KUKA KRL program: EPS_2_25694_GD01_A_20260114065858.src

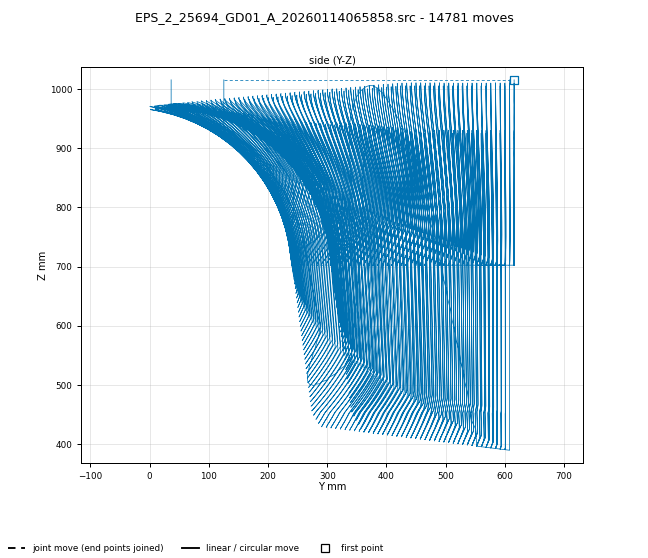
[picture p0: tool path of EPS_2_25694_GD01_A_20260114065858.src, 14781 of 14783 moves have a stored position in this frame; points joined in program order, loops and branches not executed]
&ACCESS RVP
&REL 4
&COMMENT QRS 19112012
&PARAM EDITMASK = *
DEF PART()
EXT BAS (BAS_COMMAND :IN,REAL :IN )
INT I
BAS (#INITMOV,0 )

;KUKA QRS Post kuka4.cps  Date:22-06-2017 !

File_ID=2969

QRS_PRE_INIT()

;Init var - Until changes are made in qrs_pre_init
Outlet_Square_prg=0
Inlet_1_Square_prg=0
Inlet_2_Square_prg=0
Inlet_3_Square_prg=0
Inlet_4_Square_prg=0
Inlet_5_Square_prg=0

Outlet_1={X 0.000, Y 425.000, Z 739.000, B 0.000, E1 0.000 }
Inlet_1={X 0.000, Y 466.000, Z 697.000, B 0.000, E1 153.000 }
Outlet_1_type=533
Inlet_1_type=457
;QRS#1=Sidecore dimensions
;QRS#2=525-21" Concrete
;QRS#3=450-18" Concrete
;QRS#4=
;QRS#5=
;QRS#6=
;QRS#7=
;QRS#8=
;QRS#9=S306-32
;QRS#10=28A PSX-2
;QRS#11=
;QRS#12=
;QRS#13=
;QRS#14=
;QRS#15=
;QRS#16=1220x127x1372 4,5'
;QRS#17=EPS Height
;QRS#18=1005,5
;QRS#19=*
;QRS#20= UPDATED VERSION 22-06-2017
;QRS#21=*
Outlet_Square=0250
Inlet_1_Square=0250
Inlet_2_Square=0
Inlet_3_Square=0
Inlet_4_Square=0
Inlet_5_Square=0
Mill_Square=1
Outlet_Square_Prg=263
Inlet_1_Square_prg=274

QRS_INIT()

$ADVANCE=5

; T1
PTP {E1 172.546,E2 172.546}
PTP {X 0,Y 615.562,A -85,B 0,C 180,E1 172.546,E2 172.546,E3 0,E4 0,E5 0,E6 0}
QRS_SPEED_INIT()
LIN {X 0,Y 615.562,Z 1015.5,A -85,B 0,C 180,E1 172.546,E2 172.546,E3 0,E4 0,E5 0,E6 0} C_VEL
LIN {X 0,Y 615.562,Z 704.53,A -85,B 0,C 180,E1 172.546,E2 172.546} C_VEL
LIN {X 0,Y 615.508,Z 702.53,A -85,B 0,C 180,E1 172.732,E2 172.732} C_VEL
LIN {X 0,Y 615.82,Z 702.53,A -85,B 0,C 180,E1 176.52,E2 176.52} C_VEL
LIN {X 0,Y 615.878,Z 702.53,A -85,B 0,C 180,E1 181.159,E2 181.159} C_VEL
LIN {X 0,Y 615.808,Z 702.53,A -85,B 0,C 180,E1 185.807,E2 185.807} C_VEL
LIN {X 0,Y 615.767,Z 702.53,A -85,B 0,C 180,E1 190.494,E2 190.494} C_VEL
LIN {X 0,Y 615.783,Z 702.53,A -85,B 0,C 180,E1 195.253,E2 195.253} C_VEL
LIN {X 0,Y 615.731,Z 702.53,A -85,B 0,C 180,E1 200.124,E2 200.124} C_VEL
LIN {X 0,Y 615.743,Z 702.53,A -85,B 0,C 180,E1 205.15,E2 205.15} C_VEL
LIN {X 0,Y 615.198,Z 702.53,A -85,B 0,C 180,E1 207.768,E2 207.768} C_VEL
LIN {X 0,Y 615.689,Z 702.53,A -85,B 0,C 180,E1 210.397,E2 210.397} C_VEL
LIN {X 0,Y 615.123,Z 702.53,A -85,B 0,C 180,E1 213.847,E2 213.847} C_VEL
LIN {X 0,Y 615.683,Z 702.53,A -85,B 0,C 180,E1 215.941,E2 215.941} C_VEL
LIN {X 0,Y 615.415,Z 702.53,A -85,B 0,C 180,E1 217.849,E2 217.849} C_VEL
LIN {X 0,Y 615.361,Z 702.53,A -85,B 0,C 180,E1 218.885,E2 218.885} C_VEL
LIN {X 0,Y 615.623,Z 702.53,A -85,B 0,C 180,E1 221.506,E2 221.506} C_VEL
LIN {X 0,Y 615.645,Z 702.53,A -85,B 0,C 180,E1 225.108,E2 225.108} C_VEL
LIN {X 0,Y 615.256,Z 702.53,A -85,B 0,C 180,E1 228.538,E2 228.538} C_VEL
LIN {X 0,Y 615.656,Z 702.53,A -85,B 0,C 180,E1 231.141,E2 231.141} C_VEL
LIN {X 0,Y 615.65,Z 702.53,A -85,B 0,C 180,E1 236.086,E2 236.086} C_VEL
LIN {X 0,Y 615.768,Z 702.53,A -85,B 0,C 180,E1 236.883,E2 236.883} C_VEL
LIN {X 0,Y 615.85,Z 702.53,A -85,B 0,C 180,E1 240.621,E2 240.621} C_VEL
LIN {X 0,Y 615.243,Z 702.53,A -85,B 0,C 180,E1 240.781,E2 240.781} C_VEL
LIN {X 0,Y 615.136,Z 702.999,A -85,B 0,C 180,E1 240.802,E2 240.802} C_VEL
LIN {X 0,Y 615.431,Z 753.05,A -85,B 0,C 180,E1 241.477,E2 241.477} C_VEL
LIN {X 0,Y 615.504,Z 764.124,A -85,B 0,C 180,E1 241.655,E2 241.655} C_VEL
LIN {X 0,Y 615.538,Z 778.609,A -85,B 0,C 180,E1 241.961,E2 241.961} C_VEL
LIN {X 0,Y 615.499,Z 788.804,A -85,B 0,C 180,E1 242.218,E2 242.218} C_VEL
LIN {X 0,Y 615.679,Z 804.599,A -85,B 0,C 180,E1 242.709,E2 242.709} C_VEL
LIN {X 0,Y 615.642,Z 817.021,A -85,B 0,C 180,E1 243.155,E2 243.155} C_VEL
LIN {X 0,Y 615.565,Z 826.938,A -85,B 0,C 180,E1 243.557,E2 243.557} C_VEL
LIN {X 0,Y 615.705,Z 842.65,A -85,B 0,C 180,E1 244.289,E2 244.289} C_VEL
LIN {X 0,Y 615.691,Z 854.983,A -85,B 0,C 180,E1 244.938,E2 244.938} C_VEL
LIN {X 0,Y 615.678,Z 866.612,A -85,B 0,C 180,E1 245.617,E2 245.617} C_VEL
LIN {X 0,Y 615.714,Z 878.424,A -85,B 0,C 180,E1 246.381,E2 246.381} C_VEL
LIN {X 0,Y 615.719,Z 889.118,A -85,B 0,C 180,E1 247.137,E2 247.137} C_VEL
LIN {X 0,Y 615.705,Z 900.424,A -85,B 0,C 180,E1 248.014,E2 248.014} C_VEL
LIN {X 0,Y 615.703,Z 909.682,A -85,B 0,C 180,E1 248.794,E2 248.794} C_VEL
LIN {X 0,Y 615.752,Z 919.817,A -85,B 0,C 180,E1 249.725,E2 249.725} C_VEL
LIN {X 0,Y 615.721,Z 929.079,A -85,B 0,C 180,E1 250.649,E2 250.649} C_VEL
LIN {X 0,Y 615.679,Z 937.435,A -85,B 0,C 180,E1 251.55,E2 251.55} C_VEL
LIN {X 0,Y 615.758,Z 945.796,A -85,B 0,C 180,E1 252.534,E2 252.534} C_VEL
LIN {X 0,Y 615.71,Z 953.699,A -85,B 0,C 180,E1 253.544,E2 253.544} C_VEL
LIN {X 0,Y 615.576,Z 960.443,A -85,B 0,C 180,E1 254.475,E2 254.475} C_VEL
LIN {X 0,Y 615.669,Z 968.075,A -85,B 0,C 180,E1 255.647,E2 255.647} C_VEL
LIN {X 0,Y 615.808,Z 973.451,A -85,B 0,C 180,E1 256.546,E2 256.546} C_VEL
LIN {X 0,Y 615.571,Z 979.922,A -85,B 0,C 180,E1 257.73,E2 257.73} C_VEL
LIN {X 0,Y 615.608,Z 985.635,A -85,B 0,C 180,E1 258.915,E2 258.915} C_VEL
LIN {X 0,Y 615.819,Z 990.644,A -85,B 0,C 180,E1 260.098,E2 260.098} C_VEL
LIN {X 0,Y 615.602,Z 995.072,A -85,B 0,C 180,E1 261.27,E2 261.27} C_VEL
LIN {X 0,Y 615.662,Z 999.448,A -85,B 0,C 180,E1 262.653,E2 262.653} C_VEL
LIN {X 0,Y 615.802,Z 1002.367,A -85,B 0,C 180,E1 263.749,E2 263.749} C_VEL
LIN {X 0,Y 615.545,Z 1005.385,A -85,B 0,C 180,E1 265.125,E2 265.125} C_VEL
LIN {X 0,Y 615.635,Z 1007.595,A -85,B 0,C 180,E1 266.521,E2 266.521} C_VEL
LIN {X 0,Y 615.819,Z 1008.672,A -85,B 0,C 180,E1 267.451,E2 267.451} C_VEL
LIN {X 0,Y 615.544,Z 1009.717,A -85,B 0,C 180,E1 268.842,E2 268.842} C_VEL
LIN {X 0,Y 615.843,Z 1009.658,A -85,B 0,C 180,E1 271.162,E2 271.162} C_VEL
LIN {X 0,Y 615.558,Z 1008.716,A -85,B 0,C 180,E1 272.555,E2 272.555} C_VEL
LIN {X 0,Y 615.598,Z 1006.932,A -85,B 0,C 180,E1 273.949,E2 273.949} C_VEL
LIN {X 0,Y 615.806,Z 1005.329,A -85,B 0,C 180,E1 274.878,E2 274.878} C_VEL
LIN {X 0,Y 615.606,Z 1002.401,A -85,B 0,C 180,E1 276.253,E2 276.253} C_VEL
LIN {X 0,Y 615.625,Z 999.259,A -85,B 0,C 180,E1 277.421,E2 277.421} C_VEL
LIN {X 0,Y 615.798,Z 995.025,A -85,B 0,C 180,E1 278.732,E2 278.732} C_VEL
LIN {X 0,Y 615.583,Z 990.661,A -85,B 0,C 180,E1 279.91,E2 279.91} C_VEL
LIN {X 0,Y 615.638,Z 985.611,A -85,B 0,C 180,E1 281.089,E2 281.089} C_VEL
LIN {X 0,Y 615.808,Z 979.871,A -85,B 0,C 180,E1 282.269,E2 282.269} C_VEL
LIN {X 0,Y 615.627,Z 973.442,A -85,B 0,C 180,E1 283.463,E2 283.463} C_VEL
LIN {X 0,Y 615.697,Z 966.18,A -85,B 0,C 180,E1 284.656,E2 284.656} C_VEL
LIN {X 0,Y 615.81,Z 960.631,A -85,B 0,C 180,E1 285.488,E2 285.488} C_VEL
LIN {X 0,Y 615.662,Z 951.188,A -85,B 0,C 180,E1 286.792,E2 286.792} C_VEL
LIN {X 0,Y 615.738,Z 942.596,A -85,B 0,C 180,E1 287.853,E2 287.853} C_VEL
LIN {X 0,Y 615.77,Z 934.395,A -85,B 0,C 180,E1 288.786,E2 288.786} C_VEL
LIN {X 0,Y 615.695,Z 924.501,A -85,B 0,C 180,E1 289.818,E2 289.818} C_VEL
LIN {X 0,Y 615.712,Z 916.513,A -85,B 0,C 180,E1 290.59,E2 290.59} C_VEL
LIN {X 0,Y 615.743,Z 906.008,A -85,B 0,C 180,E1 291.521,E2 291.521} C_VEL
LIN {X 0,Y 615.702,Z 896.053,A -85,B 0,C 180,E1 292.335,E2 292.335} C_VEL
LIN {X 0,Y 615.701,Z 886.27,A -85,B 0,C 180,E1 293.073,E2 293.073} C_VEL
LIN {X 0,Y 615.683,Z 874.62,A -85,B 0,C 180,E1 293.874,E2 293.874} C_VEL
LIN {X 0,Y 615.687,Z 862.583,A -85,B 0,C 180,E1 294.624,E2 294.624} C_VEL
LIN {X 0,Y 615.65,Z 851.845,A -85,B 0,C 180,E1 295.236,E2 295.236} C_VEL
LIN {X 0,Y 615.643,Z 840.977,A -85,B 0,C 180,E1 295.799,E2 295.799} C_VEL
LIN {X 0,Y 615.698,Z 826.817,A -85,B 0,C 180,E1 296.442,E2 296.442} C_VEL
LIN {X 0,Y 615.612,Z 813.606,A -85,B 0,C 180,E1 296.973,E2 296.973} C_VEL
LIN {X 0,Y 615.554,Z 804.458,A -85,B 0,C 180,E1 297.302,E2 297.302} C_VEL
LIN {X 0,Y 615.621,Z 787.798,A -85,B 0,C 180,E1 297.802,E2 297.802} C_VEL
LIN {X 0,Y 615.444,Z 775.356,A -85,B 0,C 180,E1 298.119,E2 298.119} C_VEL
LIN {X 0,Y 615.619,Z 763.086,A -85,B 0,C 180,E1 298.358,E2 298.358} C_VEL
LIN {X 0,Y 615.529,Z 741.859,A -85,B 0,C 180,E1 298.67,E2 298.67} C_VEL
LIN {X 0,Y 615.156,Z 705.781,A -85,B 0,C 180,E1 299.16,E2 299.16} C_VEL
LIN {X 0,Y 615.189,Z 702.53,A -85,B 0,C 180,E1 299.214,E2 299.214} C_VEL
LIN {X 0,Y 615.793,Z 702.53,A -85,B 0,C 180,E1 299.348,E2 299.348} C_VEL
LIN {X 0,Y 615.858,Z 702.53,A -85,B 0,C 180,E1 300.389,E2 300.389} C_VEL
LIN {X 0,Y 615.142,Z 702.53,A -85,B 0,C 180,E1 303.843,E2 303.843} C_VEL
LIN {X 0,Y 615.684,Z 702.53,A -85,B 0,C 180,E1 305.943,E2 305.943} C_VEL
LIN {X 0,Y 615.413,Z 702.53,A -85,B 0,C 180,E1 307.842,E2 307.842} C_VEL
LIN {X 0,Y 615.368,Z 702.53,A -85,B 0,C 180,E1 308.886,E2 308.886} C_VEL
LIN {X 0,Y 615.646,Z 702.53,A -85,B 0,C 180,E1 311.503,E2 311.503} C_VEL
LIN {X 0,Y 615.676,Z 702.53,A -85,B 0,C 180,E1 315.106,E2 315.106} C_VEL
LIN {X 0,Y 615.268,Z 702.53,A -85,B 0,C 180,E1 318.538,E2 318.538} C_VEL
LIN {X 0,Y 615.647,Z 702.53,A -85,B 0,C 180,E1 321.136,E2 321.136} C_VEL
LIN {X 0,Y 615.643,Z 702.53,A -85,B 0,C 180,E1 326.089,E2 326.089} C_VEL
LIN {X 0,Y 615.727,Z 702.53,A -85,B 0,C 180,E1 326.877,E2 326.877} C_VEL
LIN {X 0,Y 615.545,Z 702.53,A -85,B 0,C 180,E1 330.519,E2 330.519} C_VEL
LIN {X 0,Y 615.511,Z 702.53,A -85,B 0,C 180,E1 332.248,E2 332.248} C_VEL
LIN {X 0,Y 615.444,Z 702.53,A -85,B 0,C 180,E1 335.666,E2 335.666} C_VEL
LIN {X 0,Y 615.603,Z 702.53,A -85,B 0,C 180,E1 337.381,E2 337.381} C_VEL
LIN {X 0,Y 615.792,Z 702.53,A -85,B 0,C 180,E1 342.011,E2 342.011} C_VEL
LIN {X 0,Y 615.795,Z 702.53,A -85,B 0,C 180,E1 342.329,E2 342.329} C_VEL
LIN {X 0,Y 615.806,Z 702.53,A -85,B 0,C 180,E1 347.139,E2 347.139} C_VEL
LIN {X 0,Y 615.843,Z 702.53,A -85,B 0,C 180,E1 351.857,E2 351.857} C_VEL
LIN {X 0,Y 615.853,Z 702.53,A -85,B 0,C 180,E1 356.52,E2 356.52} C_VEL
LIN {X 0,Y 615.874,Z 702.53,A -85,B 0,C 180,E1 361.159,E2 361.159} C_VEL
LIN {X 0,Y 615.853,Z 702.53,A -85,B 0,C 180,E1 365.807,E2 365.807} C_VEL
LIN {X 0,Y 615.827,Z 702.53,A -85,B 0,C 180,E1 370.493,E2 370.493} C_VEL
LIN {X 0,Y 615.802,Z 702.53,A -85,B 0,C 180,E1 375.252,E2 375.252} C_VEL
LIN {X 0,Y 615.774,Z 702.53,A -85,B 0,C 180,E1 380.122,E2 380.122} C_VEL
LIN {X 0,Y 615.742,Z 702.53,A -85,B 0,C 180,E1 385.151,E2 385.151} C_VEL
LIN {X 0,Y 615.393,Z 702.53,A -85,B 0,C 180,E1 389.456,E2 389.456} C_VEL
LIN {X 0,Y 615.722,Z 702.53,A -85,B 0,C 180,E1 390.395,E2 390.395} C_VEL
LIN {X 0,Y 615.139,Z 702.53,A -85,B 0,C 180,E1 393.841,E2 393.841} C_VEL
LIN {X 0,Y 615.684,Z 702.53,A -85,B 0,C 180,E1 395.941,E2 395.941} C_VEL
LIN {X 0,Y 615.422,Z 702.53,A -85,B 0,C 180,E1 397.842,E2 397.842} C_VEL
LIN {X 0,Y 615.37,Z 702.53,A -85,B 0,C 180,E1 398.885,E2 398.885} C_VEL
LIN {X 0,Y 615.653,Z 702.53,A -85,B 0,C 180,E1 401.502,E2 401.502} C_VEL
LIN {X 0,Y 615.678,Z 702.53,A -85,B 0,C 180,E1 405.105,E2 405.105} C_VEL
LIN {X 0,Y 615.261,Z 702.53,A -85,B 0,C 180,E1 408.538,E2 408.538} C_VEL
LIN {X 0,Y 615.649,Z 702.53,A -85,B 0,C 180,E1 411.135,E2 411.135} C_VEL
LIN {X 0,Y 615.652,Z 702.53,A -85,B 0,C 180,E1 416.086,E2 416.086} C_VEL
LIN {X 0,Y 615.727,Z 702.53,A -85,B 0,C 180,E1 416.876,E2 416.876} C_VEL
LIN {X 0,Y 615.542,Z 702.53,A -85,B 0,C 180,E1 420.519,E2 420.519} C_VEL
LIN {X 0,Y 615.51,Z 702.53,A -85,B 0,C 180,E1 422.246,E2 422.246} C_VEL
LIN {X 0,Y 615.439,Z 702.53,A -85,B 0,C 180,E1 425.666,E2 425.666} C_VEL
LIN {X 0,Y 615.604,Z 702.53,A -85,B 0,C 180,E1 427.379,E2 427.379} C_VEL
LIN {X 0,Y 615.783,Z 702.53,A -85,B 0,C 180,E1 432.012,E2 432.012} C_VEL
LIN {X 0,Y 615.784,Z 702.53,A -85,B 0,C 180,E1 432.327,E2 432.327} C_VEL
LIN {X 0,Y 615.823,Z 702.53,A -85,B 0,C 180,E1 437.137,E2 437.137} C_VEL
LIN {X 0,Y 615.848,Z 702.53,A -85,B 0,C 180,E1 441.855,E2 441.855} C_VEL
LIN {X 0,Y 615.872,Z 702.53,A -85,B 0,C 180,E1 446.518,E2 446.518} C_VEL
LIN {X 0,Y 615.841,Z 702.53,A -85,B 0,C 180,E1 451.978,E2 451.978} C_VEL
LIN {X 0,Y 615.751,Z 702.53,A -85,B 0,C 180,E1 452.139,E2 452.139} C_VEL
LIN {X 0,Y 615.083,Z 702.53,A -85,B 0,C 180,E1 452.275,E2 452.275} C_VEL
LIN {X 0,Y 615.009,Z 702.774,A -85,B 0,C 180,E1 452.289,E2 452.289} C_VEL
LIN {X 0,Y 615.473,Z 717.375,A -85,B 0,C 180,E1 452.535,E2 452.535} C_VEL
LIN {X 0,Y 615.547,Z 729.182,A -85,B 0,C 180,E1 452.782,E2 452.782} C_VEL
LIN {X 0,Y 615.679,Z 740.947,A -85,B 0,C 180,E1 453.09,E2 453.09} C_VEL
LIN {X 0,Y 615.661,Z 751.951,A -85,B 0,C 180,E1 453.425,E2 453.425} C_VEL
LIN {X 0,Y 615.661,Z 761.787,A -85,B 0,C 180,E1 453.769,E2 453.769} C_VEL
LIN {X 0,Y 615.74,Z 774.534,A -85,B 0,C 180,E1 454.292,E2 454.292} C_VEL
LIN {X 0,Y 615.724,Z 784.661,A -85,B 0,C 180,E1 454.757,E2 454.757} C_VEL
LIN {X 0,Y 615.705,Z 794.885,A -85,B 0,C 180,E1 455.281,E2 455.281} C_VEL
LIN {X 0,Y 615.757,Z 806.034,A -85,B 0,C 180,E1 455.923,E2 455.923} C_VEL
LIN {X 0,Y 615.746,Z 815.383,A -85,B 0,C 180,E1 456.513,E2 456.513} C_VEL
LIN {X 0,Y 615.752,Z 824.921,A -85,B 0,C 180,E1 457.175,E2 457.175} C_VEL
LIN {X 0,Y 615.745,Z 833.623,A -85,B 0,C 180,E1 457.832,E2 457.832} C_VEL
LIN {X 0,Y 615.768,Z 842.678,A -85,B 0,C 180,E1 458.581,E2 458.581} C_VEL
LIN {X 0,Y 615.77,Z 850.852,A -85,B 0,C 180,E1 459.314,E2 459.314} C_VEL
LIN {X 0,Y 615.719,Z 859.842,A -85,B 0,C 180,E1 460.198,E2 460.198} C_VEL
LIN {X 0,Y 615.732,Z 866.741,A -85,B 0,C 180,E1 460.935,E2 460.935} C_VEL
LIN {X 0,Y 615.825,Z 874.318,A -85,B 0,C 180,E1 461.82,E2 461.82} C_VEL
LIN {X 0,Y 615.693,Z 881.358,A -85,B 0,C 180,E1 462.713,E2 462.713} C_VEL
LIN {X 0,Y 615.672,Z 887.77,A -85,B 0,C 180,E1 463.606,E2 463.606} C_VEL
LIN {X 0,Y 615.768,Z 892.697,A -85,B 0,C 180,E1 464.351,E2 464.351} C_VEL
LIN {X 0,Y 615.762,Z 898.133,A -85,B 0,C 180,E1 465.25,E2 465.25} C_VEL
LIN {X 0,Y 615.658,Z 904.637,A -85,B 0,C 180,E1 466.457,E2 466.457} C_VEL
LIN {X 0,Y 615.722,Z 908.539,A -85,B 0,C 180,E1 467.264,E2 467.264} C_VEL
LIN {X 0,Y 615.79,Z 911.864,A -85,B 0,C 180,E1 468.039,E2 468.039} C_VEL
LIN {X 0,Y 615.662,Z 915.248,A -85,B 0,C 180,E1 468.893,E2 468.893} C_VEL
LIN {X 0,Y 615.645,Z 917.494,A -85,B 0,C 180,E1 469.507,E2 469.507} C_VEL
LIN {X 0,Y 615.809,Z 921.259,A -85,B 0,C 180,E1 470.737,E2 470.737} C_VEL
LIN {X 0,Y 615.659,Z 924.082,A -85,B 0,C 180,E1 471.83,E2 471.83} C_VEL
LIN {X 0,Y 615.578,Z 925.81,A -85,B 0,C 180,E1 472.617,E2 472.617} C_VEL
LIN {X 0,Y 615.655,Z 927.35,A -85,B 0,C 180,E1 473.537,E2 473.537} C_VEL
LIN {X 0,Y 615.833,Z 928.448,A -85,B 0,C 180,E1 474.415,E2 474.415} C_VEL
LIN {X 0,Y 615.672,Z 929.19,A -85,B 0,C 180,E1 475.15,E2 475.15} C_VEL
LIN {X 0,Y 615.566,Z 929.862,A -85,B 0,C 180,E1 476.443,E2 476.443} C_VEL
LIN {X 0,Y 615.629,Z 929.941,A -85,B 0,C 180,E1 477.09,E2 477.09} C_VEL
LIN {X 0,Y 615.759,Z 929.762,A -85,B 0,C 180,E1 477.737,E2 477.737} C_VEL
LIN {X 0,Y 615.724,Z 929.269,A -85,B 0,C 180,E1 478.633,E2 478.633} C_VEL
LIN {X 0,Y 615.654,Z 928.477,A -85,B 0,C 180,E1 479.5,E2 479.5} C_VEL
LIN {X 0,Y 615.725,Z 927.304,A -85,B 0,C 180,E1 480.392,E2 480.392} C_VEL
LIN {X 0,Y 615.769,Z 925.725,A -85,B 0,C 180,E1 481.316,E2 481.316} C_VEL
LIN {X 0,Y 615.604,Z 923.699,A -85,B 0,C 180,E1 482.262,E2 482.262} C_VEL
LIN {X 0,Y 615.648,Z 920.259,A -85,B 0,C 180,E1 483.54,E2 483.54} C_VEL
LIN {X 0,Y 615.84,Z 917.349,A -85,B 0,C 180,E1 484.436,E2 484.436} C_VEL
LIN {X 0,Y 615.648,Z 912.677,A -85,B 0,C 180,E1 485.689,E2 485.689} C_VEL
LIN {X 0,Y 615.667,Z 908.205,A -85,B 0,C 180,E1 486.717,E2 486.717} C_VEL
LIN {X 0,Y 615.805,Z 904.101,A -85,B 0,C 180,E1 487.557,E2 487.557} C_VEL
LIN {X 0,Y 615.688,Z 898.359,A -85,B 0,C 180,E1 488.624,E2 488.624} C_VEL
LIN {X 0,Y 615.655,Z 891.34,A -85,B 0,C 180,E1 489.77,E2 489.77} C_VEL
LIN {X 0,Y 615.809,Z 884.46,A -85,B 0,C 180,E1 490.771,E2 490.771} C_VEL
LIN {X 0,Y 615.739,Z 877.668,A -85,B 0,C 180,E1 491.676,E2 491.676} C_VEL
LIN {X 0,Y 615.707,Z 871.255,A -85,B 0,C 180,E1 492.461,E2 492.461} C_VEL
LIN {X 0,Y 615.792,Z 862.791,A -85,B 0,C 180,E1 493.401,E2 493.401} C_VEL
LIN {X 0,Y 615.748,Z 855.188,A -85,B 0,C 180,E1 494.178,E2 494.178} C_VEL
LIN {X 0,Y 615.734,Z 846.42,A -85,B 0,C 180,E1 494.998,E2 494.998} C_VEL
LIN {X 0,Y 615.76,Z 839.129,A -85,B 0,C 180,E1 495.628,E2 495.628} C_VEL
LIN {X 0,Y 615.759,Z 830.678,A -85,B 0,C 180,E1 496.305,E2 496.305} C_VEL
LIN {X 0,Y 615.759,Z 821.705,A -85,B 0,C 180,E1 496.965,E2 496.965} C_VEL
LIN {X 0,Y 615.741,Z 811.832,A -85,B 0,C 180,E1 497.628,E2 497.628} C_VEL
LIN {X 0,Y 615.677,Z 800.964,A -85,B 0,C 180,E1 498.288,E2 498.288} C_VEL
LIN {X 0,Y 615.74,Z 791.443,A -85,B 0,C 180,E1 498.81,E2 498.81} C_VEL
LIN {X 0,Y 615.724,Z 780.829,A -85,B 0,C 180,E1 499.335,E2 499.335} C_VEL
LIN {X 0,Y 615.617,Z 771.032,A -85,B 0,C 180,E1 499.776,E2 499.776} C_VEL
LIN {X 0,Y 615.727,Z 759.41,A -85,B 0,C 180,E1 500.225,E2 500.225} C_VEL
LIN {X 0,Y 615.68,Z 746.955,A -85,B 0,C 180,E1 500.643,E2 500.643} C_VEL
LIN {X 0,Y 615.636,Z 737.302,A -85,B 0,C 180,E1 500.925,E2 500.925} C_VEL
LIN {X 0,Y 615.748,Z 724.036,A -85,B 0,C 180,E1 501.232,E2 501.232} C_VEL
LIN {X 0,Y 615.713,Z 712.712,A -85,B 0,C 180,E1 501.445,E2 501.445} C_VEL
LIN {X 0,Y 615.553,Z 702.53,A -85,B 0,C 180,E1 501.611,E2 501.611} C_VEL
LIN {X 0,Y 615.879,Z 702.53,A -85,B 0,C 180,E1 501.784,E2 501.784} C_VEL
LIN {X 0,Y 615.704,Z 702.53,A -85,B 0,C 180,E1 504.06,E2 504.06} C_VEL
LIN {X 0,Y 615.141,Z 702.53,A -85,B 0,C 180,E1 506.841,E2 506.841} C_VEL
LIN {X 0,Y 615.715,Z 702.53,A -85,B 0,C 180,E1 509.604,E2 509.604} C_VEL
LIN {X 0,Y 615.223,Z 702.53,A -85,B 0,C 180,E1 512.234,E2 512.234} C_VEL
LIN {X 0,Y 615.765,Z 702.53,A -85,B 0,C 180,E1 514.851,E2 514.851} C_VEL
LIN {X 0,Y 615.778,Z 702.53,A -85,B 0,C 180,E1 519.878,E2 519.878} C_VEL
LIN {X 0,Y 615.518,Z 702.53,A -85,B 0,C 180,E1 522.321,E2 522.321} C_VEL
LIN {X 0,Y 615.631,Z 702.53,A -85,B 0,C 180,E1 524.743,E2 524.743} C_VEL
LIN {X 0,Y 615.831,Z 702.53,A -85,B 0,C 180,E1 527.139,E2 527.139} C_VEL
LIN {X 0,Y 615.803,Z 702.53,A -85,B 0,C 180,E1 531.857,E2 531.857} C_VEL
LIN {X 0,Y 615.508,Z 702.53,A -85,B 0,C 180,E1 532.732,E2 532.732} C_VEL
LIN {X 0,Y 611.504,Z 702.53,A -85,B 0,C 180,E1 534.32,E2 534.32} C_VEL
LIN {X 0,Y 607.646,Z 702.53,A -85,B 0,C 180,E1 535.927,E2 535.927} C_VEL
LIN {X 0,Y 607.882,Z 702.53,A -85,B 0,C 180,E1 541.434,E2 541.434} C_VEL
LIN {X 0,Y 607.632,Z 702.53,A -85,B 0,C 180,E1 546.594,E2 546.594} C_VEL
LIN {X 0,Y 607.527,Z 702.53,A -85,B 0,C 180,E1 551.47,E2 551.47} C_VEL
LIN {X 0,Y 607.63,Z 702.53,A -85,B 0,C 180,E1 555.862,E2 555.862} C_VEL
LIN {X 0,Y 607.744,Z 702.53,A -85,B 0,C 180,E1 560.349,E2 560.349} C_VEL
LIN {X 0,Y 607.769,Z 702.53,A -85,B 0,C 180,E1 564.973,E2 564.973} C_VEL
LIN {X 0,Y 607.567,Z 702.53,A -85,B 0,C 180,E1 569.79,E2 569.79} C_VEL
LIN {X 0,Y 607.62,Z 702.53,A -85,B 0,C 180,E1 576.591,E2 576.591} C_VEL
LIN {X 0,Y 607.565,Z 702.53,A -85,B 0,C 180,E1 582.117,E2 582.117} C_VEL
LIN {X 0,Y 607.258,Z 702.53,A -85,B 0,C 180,E1 587.86,E2 587.86} C_VEL
LIN {X 0,Y 607.289,Z 702.53,A -85,B 0,C 180,E1 592.671,E2 592.671} C_VEL
LIN {X 0,Y 607.695,Z 702.53,A -85,B 0,C 180,E1 597.595,E2 597.595} C_VEL
LIN {X 0,Y 607.882,Z 702.53,A -85,B 0,C 180,E1 600.411,E2 600.411} C_VEL
LIN {X 0,Y 608.572,Z 775.577,A -85,B 0,C 180,E1 601.539,E2 601.539} C_VEL
LIN {X 0,Y 608.562,Z 814.928,A -85,B 0,C 180,E1 602.736,E2 602.736} C_VEL
LIN {X 0,Y 608.415,Z 852.42,A -85,B 0,C 180,E1 604.472,E2 604.472} C_VEL
LIN {X 0,Y 608.266,Z 888.674,A -85,B 0,C 180,E1 606.806,E2 606.806} C_VEL
LIN {X 0,Y 608.119,Z 920.038,A -85,B 0,C 180,E1 609.481,E2 609.481} C_VEL
LIN {X 0,Y 608.016,Z 947.232,A -85,B 0,C 180,E1 612.486,E2 612.486} C_VEL
LIN {X 0,Y 607.884,Z 970.252,A -85,B 0,C 180,E1 615.81,E2 615.81} C_VEL
LIN {X 0,Y 607.811,Z 987.976,A -85,B 0,C 180,E1 619.268,E2 619.268} C_VEL
LIN {X 0,Y 607.799,Z 1000.677,A -85,B 0,C 180,E1 622.869,E2 622.869} C_VEL
LIN {X 0,Y 607.67,Z 1006.955,A -85,B 0,C 180,E1 625.727,E2 625.727} C_VEL
LIN {X 0,Y 607.699,Z 1010.085,A -85,B 0,C 180,E1 628.577,E2 628.577} C_VEL
LIN {X 0,Y 607.885,Z 1010.086,A -85,B 0,C 180,E1 631.422,E2 631.422} C_VEL
LIN {X 0,Y 607.905,Z 1005.757,A -85,B 0,C 180,E1 634.984,E2 634.984} C_VEL
LIN {X 0,Y 607.892,Z 995.072,A -85,B 0,C 180,E1 638.925,E2 638.925} C_VEL
LIN {X 0,Y 607.908,Z 979.45,A -85,B 0,C 180,E1 642.545,E2 642.545} C_VEL
LIN {X 0,Y 607.957,Z 958.349,A -85,B 0,C 180,E1 646.03,E2 646.03} C_VEL
LIN {X 0,Y 608.033,Z 932.214,A -85,B 0,C 180,E1 649.268,E2 649.268} C_VEL
LIN {X 0,Y 608.17,Z 902.022,A -85,B 0,C 180,E1 652.138,E2 652.138} C_VEL
LIN {X 0,Y 608.309,Z 868.887,A -85,B 0,C 180,E1 654.552,E2 654.552} C_VEL
LIN {X 0,Y 608.48,Z 832.739,A -85,B 0,C 180,E1 656.513,E2 656.513} C_VEL
LIN {X 0,Y 608.589,Z 795.74,A -85,B 0,C 180,E1 657.917,E2 657.917} C_VEL
LIN {X 0,Y 608.661,Z 760.101,A -85,B 0,C 180,E1 658.759,E2 658.759} C_VEL
LIN {X 0,Y 607.904,Z 702.53,A -85,B 0,C 180,E1 659.587,E2 659.587} C_VEL
LIN {X 0,Y 607.619,Z 702.53,A -85,B 0,C 180,E1 666.587,E2 666.587} C_VEL
LIN {X 0,Y 607.606,Z 702.53,A -85,B 0,C 180,E1 672.11,E2 672.11} C_VEL
LIN {X 0,Y 607.275,Z 702.53,A -85,B 0,C 180,E1 677.858,E2 677.858} C_VEL
LIN {X 0,Y 607.28,Z 702.53,A -85,B 0,C 180,E1 682.671,E2 682.671} C_VEL
LIN {X 0,Y 607.588,Z 702.53,A -85,B 0,C 180,E1 687.611,E2 687.611} C_VEL
LIN {X 0,Y 607.59,Z 702.53,A -85,B 0,C 180,E1 691.837,E2 691.837} C_VEL
LIN {X 0,Y 607.473,Z 702.53,A -85,B 0,C 180,E1 698.116,E2 698.116} C_VEL
LIN {X 0,Y 607.777,Z 702.53,A -85,B 0,C 180,E1 702.658,E2 702.658} C_VEL
LIN {X 0,Y 607.875,Z 702.53,A -85,B 0,C 180,E1 707.081,E2 707.081} C_VEL
LIN {X 0,Y 607.617,Z 702.53,A -85,B 0,C 180,E1 712.857,E2 712.857} C_VEL
LIN {X 0,Y 607.732,Z 702.53,A -85,B 0,C 180,E1 717.143,E2 717.143} C_VEL
LIN {X 0,Y 607.869,Z 702.53,A -85,B 0,C 180,E1 721.411,E2 721.411} C_VEL
LIN {X 0,Y 607.675,Z 702.53,A -85,B 0,C 180,E1 726.632,E2 726.632} C_VEL
LIN {X 0,Y 607.598,Z 702.53,A -85,B 0,C 180,E1 731.446,E2 731.446} C_VEL
LIN {X 0,Y 607.677,Z 702.53,A -85,B 0,C 180,E1 735.837,E2 735.837} C_VEL
LIN {X 0,Y 607.78,Z 702.53,A -85,B 0,C 180,E1 740.323,E2 740.323} C_VEL
LIN {X 0,Y 607.769,Z 702.53,A -85,B 0,C 180,E1 744.948,E2 744.948} C_VEL
LIN {X 0,Y 607.595,Z 702.53,A -85,B 0,C 180,E1 749.762,E2 749.762} C_VEL
LIN {X 0,Y 607.624,Z 702.53,A -85,B 0,C 180,E1 756.562,E2 756.562} C_VEL
LIN {X 0,Y 607.609,Z 702.53,A -85,B 0,C 180,E1 762.082,E2 762.082} C_VEL
LIN {X 0,Y 607.29,Z 702.53,A -85,B 0,C 180,E1 767.863,E2 767.863} C_VEL
LIN {X 0,Y 607.288,Z 702.53,A -85,B 0,C 180,E1 772.633,E2 772.633} C_VEL
LIN {X 0,Y 607.599,Z 702.53,A -85,B 0,C 180,E1 777.567,E2 777.567} C_VEL
LIN {X 0,Y 607.58,Z 702.53,A -85,B 0,C 180,E1 781.843,E2 781.843} C_VEL
LIN {X 0,Y 607.491,Z 702.53,A -85,B 0,C 180,E1 788.124,E2 788.124} C_VEL
LIN {X 0,Y 607.741,Z 702.53,A -85,B 0,C 180,E1 792.665,E2 792.665} C_VEL
LIN {X 0,Y 607.896,Z 702.53,A -85,B 0,C 180,E1 797.091,E2 797.091} C_VEL
LIN {X 0,Y 607.622,Z 702.53,A -85,B 0,C 180,E1 802.867,E2 802.867} C_VEL
LIN {X 0,Y 607.686,Z 702.53,A -85,B 0,C 180,E1 807.153,E2 807.153} C_VEL
LIN {X 0,Y 607.944,Z 702.53,A -85,B 0,C 180,E1 811.956,E2 811.956} C_VEL
LIN {X 0,Y 608.422,Z 742.827,A -85,B 0,C 180,E1 812.843,E2 812.843} C_VEL
LIN {X 0,Y 608.35,Z 776.479,A -85,B 0,C 180,E1 814.09,E2 814.09} C_VEL
LIN {X 0,Y 608.247,Z 809.586,A -85,B 0,C 180,E1 815.874,E2 815.874} C_VEL
LIN {X 0,Y 608.108,Z 841.848,A -85,B 0,C 180,E1 818.266,E2 818.266} C_VEL
LIN {X 0,Y 607.975,Z 869.921,A -85,B 0,C 180,E1 821.091,E2 821.091} C_VEL
LIN {X 0,Y 607.93,Z 892.853,A -85,B 0,C 180,E1 824.189,E2 824.189} C_VEL
LIN {X 0,Y 607.864,Z 909.669,A -85,B 0,C 180,E1 827.332,E2 827.332} C_VEL
LIN {X 0,Y 607.936,Z 921.864,A -85,B 0,C 180,E1 830.715,E2 830.715} C_VEL
LIN {X 0,Y 607.78,Z 927.704,A -85,B 0,C 180,E1 833.407,E2 833.407} C_VEL
LIN {X 0,Y 607.708,Z 930.443,A -85,B 0,C 180,E1 836.681,E2 836.681} C_VEL
LIN {X 0,Y 607.783,Z 928.711,A -85,B 0,C 180,E1 839.773,E2 839.773} C_VEL
LIN {X 0,Y 607.739,Z 922.093,A -85,B 0,C 180,E1 843.111,E2 843.111} C_VEL
LIN {X 0,Y 607.795,Z 911.669,A -85,B 0,C 180,E1 846.109,E2 846.109} C_VEL
LIN {X 0,Y 607.806,Z 895.517,A -85,B 0,C 180,E1 849.279,E2 849.279} C_VEL
LIN {X 0,Y 607.951,Z 874.115,A -85,B 0,C 180,E1 852.321,E2 852.321} C_VEL
LIN {X 0,Y 608.077,Z 847.473,A -85,B 0,C 180,E1 855.139,E2 855.139} C_VEL
LIN {X 0,Y 608.19,Z 817.921,A -85,B 0,C 180,E1 857.487,E2 857.487} C_VEL
LIN {X 0,Y 608.323,Z 784.262,A -85,B 0,C 180,E1 859.458,E2 859.458} C_VEL
LIN {X 0,Y 608.402,Z 747.231,A -85,B 0,C 180,E1 860.936,E2 860.936} C_VEL
LIN {X 0,Y 608.502,Z 711.075,A -85,B 0,C 180,E1 861.78,E2 861.78} C_VEL
LIN {X 0,Y 607.958,Z 702.53,A -85,B 0,C 180,E1 861.946,E2 861.946} C_VEL
LIN {X 0,Y 607.444,Z 702.53,A -85,B 0,C 180,E1 868.576,E2 868.576} C_VEL
LIN {X 0,Y 607.422,Z 702.53,A -85,B 0,C 180,E1 873.457,E2 873.457} C_VEL
LIN {X 0,Y 607.315,Z 702.53,A -85,B 0,C 180,E1 876.833,E2 876.833} C_VEL
LIN {X 0,Y 607.631,Z 702.53,A -85,B 0,C 180,E1 881.181,E2 881.181} C_VEL
LIN {X 0,Y 607.936,Z 702.53,A -85,B 0,C 180,E1 887.106,E2 887.106} C_VEL
LIN {X 0,Y 607.586,Z 702.53,A -85,B 0,C 180,E1 892.88,E2 892.88} C_VEL
LIN {X 0,Y 607.646,Z 702.53,A -85,B 0,C 180,E1 895.927,E2 895.927} C_VEL
LIN {X 0,Y 606.323,Z 702.53,A -85,B 0,C 180,E1 896.741,E2 896.741} C_VEL
LIN {X 0,Y 599.65,Z 702.53,A -85,B 0,C 180,E1 898.952,E2 898.952} C_VEL
LIN {X 0,Y 599.573,Z 702.53,A -85,B 0,C 180,E1 899.162,E2 899.162} C_VEL
LIN {X 0,Y 599.624,Z 702.53,A -85,B 0,C 180,E1 902.896,E2 902.896} C_VEL
LIN {X 0,Y 599.58,Z 702.53,A -85,B 0,C 180,E1 907.239,E2 907.239} C_VEL
LIN {X 0,Y 599.601,Z 702.53,A -85,B 0,C 180,E1 911.624,E2 911.624} C_VEL
LIN {X 0,Y 599.473,Z 702.53,A -85,B 0,C 180,E1 916.95,E2 916.95} C_VEL
LIN {X 0,Y 599.53,Z 702.53,A -85,B 0,C 180,E1 921.362,E2 921.362} C_VEL
LIN {X 0,Y 599.742,Z 702.53,A -85,B 0,C 180,E1 925.331,E2 925.331} C_VEL
LIN {X 0,Y 599.488,Z 702.53,A -85,B 0,C 180,E1 931.146,E2 931.146} C_VEL
LIN {X 0,Y 599.652,Z 702.53,A -85,B 0,C 180,E1 937.158,E2 937.158} C_VEL
LIN {X 0,Y 599.551,Z 702.53,A -85,B 0,C 180,E1 943.121,E2 943.121} C_VEL
LIN {X 0,Y 599.409,Z 702.53,A -85,B 0,C 180,E1 949.114,E2 949.114} C_VEL
LIN {X 0,Y 599.307,Z 702.53,A -85,B 0,C 180,E1 953.683,E2 953.683} C_VEL
LIN {X 0,Y 599.74,Z 702.53,A -85,B 0,C 180,E1 958.103,E2 958.103} C_VEL
LIN {X 0,Y 599.864,Z 702.564,A -85,B 0,C 180,E1 959.978,E2 959.978} C_VEL
LIN {X 0,Y 601.417,Z 710.419,A -85,B 0,C 180,E1 960.169,E2 960.169} C_VEL
LIN {X 0,Y 601.6,Z 776.602,A -85,B 0,C 180,E1 961.201,E2 961.201} C_VEL
LIN {X 0,Y 601.474,Z 815.69,A -85,B 0,C 180,E1 962.416,E2 962.416} C_VEL
LIN {X 0,Y 601.133,Z 854.192,A -85,B 0,C 180,E1 964.241,E2 964.241} C_VEL
LIN {X 0,Y 600.768,Z 889.761,A -85,B 0,C 180,E1 966.585,E2 966.585} C_VEL
LIN {X 0,Y 600.495,Z 920.701,A -85,B 0,C 180,E1 969.276,E2 969.276} C_VEL
LIN {X 0,Y 600.272,Z 948.698,A -85,B 0,C 180,E1 972.442,E2 972.442} C_VEL
LIN {X 0,Y 600.065,Z 971.361,A -85,B 0,C 180,E1 975.809,E2 975.809} C_VEL
LIN {X 0,Y 599.955,Z 988.886,A -85,B 0,C 180,E1 979.343,E2 979.343} C_VEL
LIN {X 0,Y 599.899,Z 1000.677,A -85,B 0,C 180,E1 982.774,E2 982.774} C_VEL
LIN {X 0,Y 599.767,Z 1006.955,A -85,B 0,C 180,E1 985.671,E2 985.671} C_VEL
LIN {X 0,Y 599.8,Z 1010.086,A -85,B 0,C 180,E1 988.558,E2 988.558} C_VEL
LIN {X 0,Y 599.978,Z 1010.086,A -85,B 0,C 180,E1 991.441,E2 991.441} C_VEL
LIN {X 0,Y 599.993,Z 1005.757,A -85,B 0,C 180,E1 995.05,E2 995.05} C_VEL
LIN {X 0,Y 599.99,Z 995.073,A -85,B 0,C 180,E1 999.044,E2 999.044} C_VEL
LIN {X 0,Y 600.043,Z 979.451,A -85,B 0,C 180,E1 1002.712,E2 1002.712} C_VEL
LIN {X 0,Y 600.116,Z 957.721,A -85,B 0,C 180,E1 1006.333,E2 1006.333} C_VEL
LIN {X 0,Y 600.355,Z 932.069,A -85,B 0,C 180,E1 1009.541,E2 1009.541} C_VEL
LIN {X 0,Y 600.638,Z 901.462,A -85,B 0,C 180,E1 1012.478,E2 1012.478} C_VEL
LIN {X 0,Y 600.985,Z 866.931,A -85,B 0,C 180,E1 1014.999,E2 1014.999} C_VEL
LIN {X 0,Y 601.369,Z 828.903,A -85,B 0,C 180,E1 1017.033,E2 1017.033} C_VEL
LIN {X 0,Y 601.58,Z 789.536,A -85,B 0,C 180,E1 1018.464,E2 1018.464} C_VEL
LIN {X 0,Y 601.785,Z 750.404,A -85,B 0,C 180,E1 1019.273,E2 1019.273} C_VEL
LIN {X 0,Y 600.805,Z 706.091,A -85,B 0,C 180,E1 1019.922,E2 1019.922} C_VEL
LIN {X 0,Y 599.903,Z 702.53,A -85,B 0,C 180,E1 1020.023,E2 1020.023} C_VEL
LIN {X 0,Y 599.656,Z 702.53,A -85,B 0,C 180,E1 1027.154,E2 1027.154} C_VEL
LIN {X 0,Y 599.572,Z 702.53,A -85,B 0,C 180,E1 1033.121,E2 1033.121} C_VEL
LIN {X 0,Y 599.402,Z 702.53,A -85,B 0,C 180,E1 1039.11,E2 1039.11} C_VEL
LIN {X 0,Y 599.296,Z 702.53,A -85,B 0,C 180,E1 1043.683,E2 1043.683} C_VEL
LIN {X 0,Y 599.598,Z 702.53,A -85,B 0,C 180,E1 1048.09,E2 1048.09} C_VEL
LIN {X 0,Y 599.471,Z 702.53,A -85,B 0,C 180,E1 1053.051,E2 1053.051} C_VEL
LIN {X 0,Y 599.578,Z 702.53,A -85,B 0,C 180,E1 1057.813,E2 1057.813} C_VEL
LIN {X 0,Y 599.79,Z 702.53,A -85,B 0,C 180,E1 1062.95,E2 1062.95} C_VEL
LIN {X 0,Y 599.634,Z 702.53,A -85,B 0,C 180,E1 1068.376,E2 1068.376} C_VEL
LIN {X 0,Y 599.718,Z 702.53,A -85,B 0,C 180,E1 1072.762,E2 1072.762} C_VEL
LIN {X 0,Y 599.843,Z 702.53,A -85,B 0,C 180,E1 1077.105,E2 1077.105} C_VEL
LIN {X 0,Y 599.958,Z 702.53,A -85,B 0,C 180,E1 1081.429,E2 1081.429} C_VEL
LIN {X 0,Y 600.019,Z 702.53,A -85,B 0,C 180,E1 1085.761,E2 1085.761} C_VEL
LIN {X 0,Y 599.656,Z 702.53,A -85,B 0,C 180,E1 1091.599,E2 1091.599} C_VEL
LIN {X 0,Y 599.519,Z 702.53,A -85,B 0,C 180,E1 1096.966,E2 1096.966} C_VEL
LIN {X 0,Y 599.543,Z 702.53,A -85,B 0,C 180,E1 1101.366,E2 1101.366} C_VEL
LIN {X 0,Y 599.747,Z 702.53,A -85,B 0,C 180,E1 1105.305,E2 1105.305} C_VEL
LIN {X 0,Y 599.553,Z 702.53,A -85,B 0,C 180,E1 1111.157,E2 1111.157} C_VEL
LIN {X 0,Y 599.657,Z 702.53,A -85,B 0,C 180,E1 1117.129,E2 1117.129} C_VEL
LIN {X 0,Y 599.582,Z 702.53,A -85,B 0,C 180,E1 1123.125,E2 1123.125} C_VEL
LIN {X 0,Y 599.404,Z 702.53,A -85,B 0,C 180,E1 1129.114,E2 1129.114} C_VEL
LIN {X 0,Y 599.288,Z 702.53,A -85,B 0,C 180,E1 1133.646,E2 1133.646} C_VEL
LIN {X 0,Y 599.616,Z 702.53,A -85,B 0,C 180,E1 1138.096,E2 1138.096} C_VEL
LIN {X 0,Y 599.489,Z 702.53,A -85,B 0,C 180,E1 1143.058,E2 1143.058} C_VEL
LIN {X 0,Y 599.525,Z 702.53,A -85,B 0,C 180,E1 1148.572,E2 1148.572} C_VEL
LIN {X 0,Y 599.781,Z 702.53,A -85,B 0,C 180,E1 1152.869,E2 1152.869} C_VEL
LIN {X 0,Y 599.623,Z 702.53,A -85,B 0,C 180,E1 1158.385,E2 1158.385} C_VEL
LIN {X 0,Y 599.722,Z 702.53,A -85,B 0,C 180,E1 1162.773,E2 1162.773} C_VEL
LIN {X 0,Y 599.787,Z 702.53,A -85,B 0,C 180,E1 1167.116,E2 1167.116} C_VEL
LIN {X 0,Y 599.896,Z 702.599,A -85,B 0,C 180,E1 1171.622,E2 1171.622} C_VEL
LIN {X 0,Y 601.197,Z 739.287,A -85,B 0,C 180,E1 1172.428,E2 1172.428} C_VEL
LIN {X 0,Y 601.045,Z 774.178,A -85,B 0,C 180,E1 1173.689,E2 1173.689} C_VEL
LIN {X 0,Y 600.746,Z 807.985,A -85,B 0,C 180,E1 1175.496,E2 1175.496} C_VEL
LIN {X 0,Y 600.479,Z 839.921,A -85,B 0,C 180,E1 1177.854,E2 1177.854} C_VEL
LIN {X 0,Y 600.213,Z 867.857,A -85,B 0,C 180,E1 1180.638,E2 1180.638} C_VEL
LIN {X 0,Y 600.058,Z 890.372,A -85,B 0,C 180,E1 1183.637,E2 1183.637} C_VEL
LIN {X 0,Y 599.973,Z 908.36,A -85,B 0,C 180,E1 1186.915,E2 1186.915} C_VEL
LIN {X 0,Y 599.967,Z 920.514,A -85,B 0,C 180,E1 1190.154,E2 1190.154} C_VEL
LIN {X 0,Y 599.86,Z 928.284,A -85,B 0,C 180,E1 1193.735,E2 1193.735} C_VEL
LIN {X 0,Y 599.817,Z 930.498,A -85,B 0,C 180,E1 1196.927,E2 1196.927} C_VEL
LIN {X 0,Y 599.913,Z 928.249,A -85,B 0,C 180,E1 1200.204,E2 1200.204} C_VEL
LIN {X 0,Y 599.996,Z 919.917,A -85,B 0,C 180,E1 1203.945,E2 1203.945} C_VEL
LIN {X 0,Y 600.061,Z 906.675,A -85,B 0,C 180,E1 1207.348,E2 1207.348} C_VEL
LIN {X 0,Y 600.109,Z 888.587,A -85,B 0,C 180,E1 1210.546,E2 1210.546} C_VEL
LIN {X 0,Y 600.323,Z 863.839,A -85,B 0,C 180,E1 1213.725,E2 1213.725} C_VEL
LIN {X 0,Y 600.517,Z 835.883,A -85,B 0,C 180,E1 1216.393,E2 1216.393} C_VEL
LIN {X 0,Y 600.742,Z 802.992,A -85,B 0,C 180,E1 1218.729,E2 1218.729} C_VEL
LIN {X 0,Y 601.021,Z 767.23,A -85,B 0,C 180,E1 1220.518,E2 1220.518} C_VEL
LIN {X 0,Y 601.293,Z 731.494,A -85,B 0,C 180,E1 1221.68,E2 1221.68} C_VEL
LIN {X 0,Y 600.436,Z 705.055,A -85,B 0,C 180,E1 1222.229,E2 1222.229} C_VEL
LIN {X 0,Y 599.976,Z 702.53,A -85,B 0,C 180,E1 1222.357,E2 1222.357} C_VEL
LIN {X 0,Y 599.556,Z 702.53,A -85,B 0,C 180,E1 1228.843,E2 1228.843} C_VEL
LIN {X 0,Y 599.839,Z 702.53,A -85,B 0,C 180,E1 1234.913,E2 1234.913} C_VEL
LIN {X 0,Y 599.76,Z 702.53,A -85,B 0,C 180,E1 1240.925,E2 1240.925} C_VEL
LIN {X 0,Y 599.986,Z 702.53,A -85,B 0,C 180,E1 1246.932,E2 1246.932} C_VEL
LIN {X 0,Y 599.687,Z 702.53,A -85,B 0,C 180,E1 1252.785,E2 1252.785} C_VEL
LIN {X 0,Y 599.808,Z 702.53,A -85,B 0,C 180,E1 1257.128,E2 1257.128} C_VEL
LIN {X 0,Y 599.573,Z 702.53,A -85,B 0,C 180,E1 1259.162,E2 1259.162} C_VEL
LIN {X 0,Y 597.199,Z 702.53,A -85,B 0,C 180,E1 1260.397,E2 1260.397} C_VEL
LIN {X 0,Y 591.787,Z 702.53,A -85,B 0,C 180,E1 1262.459,E2 1262.459} C_VEL
LIN {X 0,Y 591.679,Z 702.53,A -85,B 0,C 180,E1 1267.336,E2 1267.336} C_VEL
LIN {X 0,Y 591.668,Z 702.53,A -85,B 0,C 180,E1 1271.782,E2 1271.782} C_VEL
LIN {X 0,Y 591.721,Z 702.53,A -85,B 0,C 180,E1 1276.3,E2 1276.3} C_VEL
LIN {X 0,Y 591.755,Z 702.53,A -85,B 0,C 180,E1 1280.924,E2 1280.924} C_VEL
LIN {X 0,Y 591.552,Z 702.53,A -85,B 0,C 180,E1 1286.768,E2 1286.768} C_VEL
LIN {X 0,Y 591.612,Z 702.53,A -85,B 0,C 180,E1 1290.679,E2 1290.679} C_VEL
LIN {X 0,Y 591.708,Z 702.53,A -85,B 0,C 180,E1 1295.918,E2 1295.918} C_VEL
LIN {X 0,Y 591.623,Z 702.53,A -85,B 0,C 180,E1 1301.546,E2 1301.546} C_VEL
LIN {X 0,Y 591.473,Z 702.53,A -85,B 0,C 180,E1 1306.461,E2 1306.461} C_VEL
LIN {X 0,Y 591.528,Z 702.53,A -85,B 0,C 180,E1 1312.265,E2 1312.265} C_VEL
LIN {X 0,Y 591.798,Z 702.53,A -85,B 0,C 180,E1 1317.623,E2 1317.623} C_VEL
LIN {X 0,Y 591.879,Z 702.668,A -85,B 0,C 180,E1 1319.532,E2 1319.532} C_VEL
LIN {X 0,Y 594.585,Z 711.49,A -85,B 0,C 180,E1 1319.806,E2 1319.806} C_VEL
LIN {X 0,Y 594.673,Z 775.135,A -85,B 0,C 180,E1 1320.802,E2 1320.802} C_VEL
LIN {X 0,Y 594.406,Z 813.799,A -85,B 0,C 180,E1 1321.988,E2 1321.988} C_VEL
LIN {X 0,Y 593.923,Z 850.551,A -85,B 0,C 180,E1 1323.701,E2 1323.701} C_VEL
LIN {X 0,Y 593.371,Z 887.104,A -85,B 0,C 180,E1 1326.066,E2 1326.066} C_VEL
LIN {X 0,Y 592.893,Z 919.833,A -85,B 0,C 180,E1 1328.909,E2 1328.909} C_VEL
LIN {X 0,Y 592.489,Z 947.234,A -85,B 0,C 180,E1 1332.012,E2 1332.012} C_VEL
LIN {X 0,Y 592.193,Z 969.163,A -85,B 0,C 180,E1 1335.237,E2 1335.237} C_VEL
LIN {X 0,Y 592.019,Z 987.282,A -85,B 0,C 180,E1 1338.81,E2 1338.81} C_VEL
LIN {X 0,Y 591.978,Z 999.717,A -85,B 0,C 180,E1 1342.309,E2 1342.309} C_VEL
LIN {X 0,Y 591.867,Z 1006.956,A -85,B 0,C 180,E1 1345.613,E2 1345.613} C_VEL
LIN {X 0,Y 591.901,Z 1010.086,A -85,B 0,C 180,E1 1348.539,E2 1348.539} C_VEL
LIN {X 0,Y 592.072,Z 1010.086,A -85,B 0,C 180,E1 1351.46,E2 1351.46} C_VEL
LIN {X 0,Y 592.093,Z 1005.757,A -85,B 0,C 180,E1 1355.118,E2 1355.118} C_VEL
LIN {X 0,Y 592.105,Z 995.073,A -85,B 0,C 180,E1 1359.165,E2 1359.165} C_VEL
LIN {X 0,Y 592.191,Z 979.451,A -85,B 0,C 180,E1 1362.883,E2 1362.883} C_VEL
LIN {X 0,Y 592.334,Z 957.954,A -85,B 0,C 180,E1 1366.521,E2 1366.521} C_VEL
LIN {X 0,Y 592.671,Z 932.009,A -85,B 0,C 180,E1 1369.811,E2 1369.811} C_VEL
LIN {X 0,Y 593.12,Z 901.758,A -85,B 0,C 180,E1 1372.754,E2 1372.754} C_VEL
LIN {X 0,Y 593.647,Z 867.736,A -85,B 0,C 180,E1 1375.277,E2 1375.277} C_VEL
LIN {X 0,Y 594.199,Z 830.633,A -85,B 0,C 180,E1 1377.304,E2 1377.304} C_VEL
LIN {X 0,Y 594.572,Z 791.806,A -85,B 0,C 180,E1 1378.76,E2 1378.76} C_VEL
LIN {X 0,Y 594.854,Z 753.957,A -85,B 0,C 180,E1 1379.591,E2 1379.591} C_VEL
LIN {X 0,Y 594.033,Z 708.555,A -85,B 0,C 180,E1 1380.265,E2 1380.265} C_VEL
LIN {X 0,Y 591.868,Z 702.53,A -85,B 0,C 180,E1 1380.516,E2 1380.516} C_VEL
LIN {X 0,Y 591.705,Z 702.53,A -85,B 0,C 180,E1 1385.914,E2 1385.914} C_VEL
LIN {X 0,Y 591.645,Z 702.53,A -85,B 0,C 180,E1 1392.295,E2 1392.295} C_VEL
LIN {X 0,Y 591.439,Z 702.53,A -85,B 0,C 180,E1 1397.724,E2 1397.724} C_VEL
LIN {X 0,Y 591.533,Z 702.53,A -85,B 0,C 180,E1 1402.262,E2 1402.262} C_VEL
LIN {X 0,Y 591.688,Z 702.53,A -85,B 0,C 180,E1 1407.612,E2 1407.612} C_VEL
LIN {X 0,Y 591.577,Z 702.53,A -85,B 0,C 180,E1 1413.227,E2 1413.227} C_VEL
LIN {X 0,Y 591.65,Z 702.53,A -85,B 0,C 180,E1 1417.499,E2 1417.499} C_VEL
LIN {X 0,Y 591.868,Z 702.53,A -85,B 0,C 180,E1 1422.177,E2 1422.177} C_VEL
LIN {X 0,Y 591.744,Z 702.53,A -85,B 0,C 180,E1 1428.219,E2 1428.219} C_VEL
LIN {X 0,Y 591.837,Z 702.53,A -85,B 0,C 180,E1 1432.666,E2 1432.666} C_VEL
LIN {X 0,Y 591.935,Z 702.53,A -85,B 0,C 180,E1 1437.066,E2 1437.066} C_VEL
LIN {X 0,Y 592.048,Z 702.53,A -85,B 0,C 180,E1 1441.448,E2 1441.448} C_VEL
LIN {X 0,Y 591.964,Z 702.53,A -85,B 0,C 180,E1 1446.185,E2 1446.185} C_VEL
LIN {X 0,Y 591.72,Z 702.53,A -85,B 0,C 180,E1 1451.757,E2 1451.757} C_VEL
LIN {X 0,Y 591.763,Z 702.53,A -85,B 0,C 180,E1 1456.274,E2 1456.274} C_VEL
LIN {X 0,Y 591.777,Z 702.53,A -85,B 0,C 180,E1 1460.898,E2 1460.898} C_VEL
LIN {X 0,Y 591.534,Z 702.53,A -85,B 0,C 180,E1 1466.765,E2 1466.765} C_VEL
LIN {X 0,Y 591.661,Z 702.53,A -85,B 0,C 180,E1 1470.649,E2 1470.649} C_VEL
LIN {X 0,Y 591.695,Z 702.53,A -85,B 0,C 180,E1 1475.89,E2 1475.89} C_VEL
LIN {X 0,Y 591.65,Z 702.53,A -85,B 0,C 180,E1 1481.512,E2 1481.512} C_VEL
LIN {X 0,Y 591.5,Z 702.53,A -85,B 0,C 180,E1 1486.463,E2 1486.463} C_VEL
LIN {X 0,Y 591.522,Z 702.53,A -85,B 0,C 180,E1 1492.247,E2 1492.247} C_VEL
LIN {X 0,Y 591.697,Z 702.53,A -85,B 0,C 180,E1 1497.618,E2 1497.618} C_VEL
LIN {X 0,Y 591.579,Z 702.53,A -85,B 0,C 180,E1 1503.174,E2 1503.174} C_VEL
LIN {X 0,Y 591.67,Z 702.53,A -85,B 0,C 180,E1 1507.507,E2 1507.507} C_VEL
LIN {X 0,Y 591.849,Z 702.53,A -85,B 0,C 180,E1 1512.184,E2 1512.184} C_VEL
LIN {X 0,Y 591.736,Z 702.53,A -85,B 0,C 180,E1 1518.228,E2 1518.228} C_VEL
LIN {X 0,Y 591.84,Z 702.53,A -85,B 0,C 180,E1 1522.676,E2 1522.676} C_VEL
LIN {X 0,Y 591.883,Z 702.53,A -85,B 0,C 180,E1 1527.077,E2 1527.077} C_VEL
LIN {X 0,Y 591.825,Z 702.53,A -85,B 0,C 180,E1 1531.233,E2 1531.233} C_VEL
LIN {X 0,Y 593.796,Z 712.995,A -85,B 0,C 180,E1 1531.502,E2 1531.502} C_VEL
LIN {X 0,Y 593.893,Z 751.831,A -85,B 0,C 180,E1 1532.503,E2 1532.503} C_VEL
LIN {X 0,Y 593.492,Z 787.156,A -85,B 0,C 180,E1 1534.01,E2 1534.01} C_VEL
LIN {X 0,Y 593.083,Z 820.796,A -85,B 0,C 180,E1 1536.08,E2 1536.08} C_VEL
LIN {X 0,Y 592.73,Z 850.826,A -85,B 0,C 180,E1 1538.602,E2 1538.602} C_VEL
LIN {X 0,Y 592.449,Z 877.324,A -85,B 0,C 180,E1 1541.592,E2 1541.592} C_VEL
LIN {X 0,Y 592.236,Z 899.248,A -85,B 0,C 180,E1 1544.951,E2 1544.951} C_VEL
LIN {X 0,Y 592.157,Z 914.214,A -85,B 0,C 180,E1 1548.19,E2 1548.19} C_VEL
LIN {X 0,Y 592.067,Z 923.99,A -85,B 0,C 180,E1 1551.368,E2 1551.368} C_VEL
LIN {X 0,Y 591.974,Z 928.723,A -85,B 0,C 180,E1 1554.071,E2 1554.071} C_VEL
LIN {X 0,Y 591.918,Z 930.425,A -85,B 0,C 180,E1 1557.316,E2 1557.316} C_VEL
LIN {X 0,Y 592.03,Z 927.621,A -85,B 0,C 180,E1 1560.649,E2 1560.649} C_VEL
LIN {X 0,Y 592.124,Z 919.72,A -85,B 0,C 180,E1 1564.102,E2 1564.102} C_VEL
LIN {X 0,Y 592.185,Z 907.34,A -85,B 0,C 180,E1 1567.346,E2 1567.346} C_VEL
LIN {X 0,Y 592.296,Z 889.279,A -85,B 0,C 180,E1 1570.621,E2 1570.621} C_VEL
LIN {X 0,Y 592.583,Z 865.208,A -85,B 0,C 180,E1 1573.801,E2 1573.801} C_VEL
LIN {X 0,Y 592.922,Z 836.23,A -85,B 0,C 180,E1 1576.623,E2 1576.623} C_VEL
LIN {X 0,Y 593.271,Z 804.415,A -85,B 0,C 180,E1 1578.929,E2 1578.929} C_VEL
LIN {X 0,Y 593.702,Z 769.297,A -85,B 0,C 180,E1 1580.741,E2 1580.741} C_VEL
LIN {X 0,Y 594.073,Z 733.605,A -85,B 0,C 180,E1 1581.947,E2 1581.947} C_VEL
LIN {X 0,Y 593.468,Z 707.373,A -85,B 0,C 180,E1 1582.511,E2 1582.511} C_VEL
LIN {X 0,Y 592.032,Z 702.53,A -85,B 0,C 180,E1 1582.685,E2 1582.685} C_VEL
LIN {X 0,Y 591.664,Z 702.53,A -85,B 0,C 180,E1 1589.352,E2 1589.352} C_VEL
LIN {X 0,Y 591.76,Z 702.53,A -85,B 0,C 180,E1 1594.329,E2 1594.329} C_VEL
LIN {X 0,Y 591.847,Z 702.53,A -85,B 0,C 180,E1 1600.66,E2 1600.66} C_VEL
LIN {X 0,Y 592.04,Z 702.53,A -85,B 0,C 180,E1 1606.754,E2 1606.754} C_VEL
LIN {X 0,Y 591.8,Z 702.53,A -85,B 0,C 180,E1 1612.716,E2 1612.716} C_VEL
LIN {X 0,Y 591.901,Z 702.53,A -85,B 0,C 180,E1 1617.09,E2 1617.09} C_VEL
LIN {X 0,Y 591.787,Z 702.53,A -85,B 0,C 180,E1 1622.459,E2 1622.459} C_VEL
LIN {X 0,Y 587.733,Z 702.53,A -85,B 0,C 180,E1 1624.115,E2 1624.115} C_VEL
LIN {X 0,Y 584.077,Z 702.53,A -85,B 0,C 180,E1 1625.794,E2 1625.794} C_VEL
LIN {X 0,Y 583.763,Z 702.53,A -85,B 0,C 180,E1 1631.944,E2 1631.944} C_VEL
LIN {X 0,Y 583.711,Z 702.53,A -85,B 0,C 180,E1 1636.954,E2 1636.954} C_VEL
LIN {X 0,Y 583.72,Z 702.53,A -85,B 0,C 180,E1 1641.46,E2 1641.46} C_VEL
LIN {X 0,Y 583.742,Z 702.53,A -85,B 0,C 180,E1 1646.076,E2 1646.076} C_VEL
LIN {X 0,Y 583.563,Z 702.53,A -85,B 0,C 180,E1 1651.423,E2 1651.423} C_VEL
LIN {X 0,Y 583.75,Z 702.53,A -85,B 0,C 180,E1 1656.739,E2 1656.739} C_VEL
LIN {X 0,Y 583.72,Z 702.53,A -85,B 0,C 180,E1 1662.237,E2 1662.237} C_VEL
LIN {X 0,Y 583.521,Z 702.53,A -85,B 0,C 180,E1 1667.749,E2 1667.749} C_VEL
LIN {X 0,Y 583.507,Z 702.53,A -85,B 0,C 180,E1 1673.294,E2 1673.294} C_VEL
LIN {X 0,Y 583.889,Z 702.53,A -85,B 0,C 180,E1 1678.525,E2 1678.525} C_VEL
LIN {X 0,Y 583.924,Z 702.53,A -85,B 0,C 180,E1 1679.044,E2 1679.044} C_VEL
LIN {X 0,Y 587.765,Z 713.889,A -85,B 0,C 180,E1 1679.452,E2 1679.452} C_VEL
LIN {X 0,Y 587.751,Z 776.602,A -85,B 0,C 180,E1 1680.456,E2 1680.456} C_VEL
LIN {X 0,Y 587.341,Z 815.781,A -85,B 0,C 180,E1 1681.697,E2 1681.697} C_VEL
LIN {X 0,Y 586.634,Z 853.696,A -85,B 0,C 180,E1 1683.526,E2 1683.526} C_VEL
LIN {X 0,Y 585.9,Z 890.027,A -85,B 0,C 180,E1 1685.975,E2 1685.975} C_VEL
LIN {X 0,Y 585.255,Z 921.947,A -85,B 0,C 180,E1 1688.84,E2 1688.84} C_VEL
LIN {X 0,Y 584.746,Z 948.7,A -85,B 0,C 180,E1 1691.96,E2 1691.96} C_VEL
LIN {X 0,Y 584.372,Z 971.571,A -85,B 0,C 180,E1 1695.456,E2 1695.456} C_VEL
LIN {X 0,Y 584.221,Z 989.852,A -85,B 0,C 180,E1 1699.289,E2 1699.289} C_VEL
LIN {X 0,Y 584.162,Z 1001.999,A -85,B 0,C 180,E1 1703.093,E2 1703.093} C_VEL
LIN {X 0,Y 584.169,Z 1008.906,A -85,B 0,C 180,E1 1707.038,E2 1707.038} C_VEL
LIN {X 0,Y 584.046,Z 1010.5,A -85,B 0,C 180,E1 1710,E2 1710} C_VEL
LIN {X 0,Y 584.022,Z 1008.907,A -85,B 0,C 180,E1 1712.962,E2 1712.962} C_VEL
LIN {X 0,Y 584.081,Z 1003.44,A -85,B 0,C 180,E1 1716.306,E2 1716.306} C_VEL
LIN {X 0,Y 584.08,Z 992.396,A -85,B 0,C 180,E1 1720.043,E2 1720.043} C_VEL
LIN {X 0,Y 584.314,Z 976.097,A -85,B 0,C 180,E1 1723.711,E2 1723.711} C_VEL
LIN {X 0,Y 584.591,Z 954.55,A -85,B 0,C 180,E1 1727.24,E2 1727.24} C_VEL
LIN {X 0,Y 585.12,Z 927.613,A -85,B 0,C 180,E1 1730.572,E2 1730.572} C_VEL
LIN {X 0,Y 585.78,Z 895.74,A -85,B 0,C 180,E1 1733.569,E2 1733.569} C_VEL
LIN {X 0,Y 586.435,Z 861.086,A -85,B 0,C 180,E1 1736.033,E2 1736.033} C_VEL
LIN {X 0,Y 587.172,Z 823.803,A -85,B 0,C 180,E1 1737.966,E2 1737.966} C_VEL
LIN {X 0,Y 587.63,Z 785.219,A -85,B 0,C 180,E1 1739.32,E2 1739.32} C_VEL
LIN {X 0,Y 587.979,Z 744.931,A -85,B 0,C 180,E1 1740.106,E2 1740.106} C_VEL
LIN {X 0,Y 587.02,Z 710.744,A -85,B 0,C 180,E1 1740.635,E2 1740.635} C_VEL
LIN {X 0,Y 583.841,Z 702.53,A -85,B 0,C 180,E1 1740.965,E2 1740.965} C_VEL
LIN {X 0,Y 583.741,Z 702.53,A -85,B 0,C 180,E1 1746.736,E2 1746.736} C_VEL
LIN {X 0,Y 583.741,Z 702.53,A -85,B 0,C 180,E1 1752.231,E2 1752.231} C_VEL
LIN {X 0,Y 583.54,Z 702.53,A -85,B 0,C 180,E1 1757.747,E2 1757.747} C_VEL
LIN {X 0,Y 583.504,Z 702.53,A -85,B 0,C 180,E1 1763.293,E2 1763.293} C_VEL
LIN {X 0,Y 583.833,Z 702.53,A -85,B 0,C 180,E1 1767.121,E2 1767.121} C_VEL
LIN {X 0,Y 583.682,Z 702.53,A -85,B 0,C 180,E1 1772.26,E2 1772.26} C_VEL
LIN {X 0,Y 583.74,Z 702.53,A -85,B 0,C 180,E1 1777.177,E2 1777.177} C_VEL
LIN {X 0,Y 583.842,Z 702.53,A -85,B 0,C 180,E1 1783.002,E2 1783.002} C_VEL
LIN {X 0,Y 583.859,Z 702.53,A -85,B 0,C 180,E1 1788.058,E2 1788.058} C_VEL
LIN {X 0,Y 583.93,Z 702.53,A -85,B 0,C 180,E1 1792.566,E2 1792.566} C_VEL
LIN {X 0,Y 584.05,Z 702.53,A -85,B 0,C 180,E1 1797.027,E2 1797.027} C_VEL
LIN {X 0,Y 584.157,Z 702.53,A -85,B 0,C 180,E1 1801.468,E2 1801.468} C_VEL
LIN {X 0,Y 584.162,Z 702.53,A -85,B 0,C 180,E1 1805.918,E2 1805.918} C_VEL
LIN {X 0,Y 583.802,Z 702.53,A -85,B 0,C 180,E1 1811.919,E2 1811.919} C_VEL
LIN {X 0,Y 583.728,Z 702.53,A -85,B 0,C 180,E1 1816.961,E2 1816.961} C_VEL
LIN {X 0,Y 583.726,Z 702.53,A -85,B 0,C 180,E1 1821.463,E2 1821.463} C_VEL
LIN {X 0,Y 583.753,Z 702.53,A -85,B 0,C 180,E1 1826.049,E2 1826.049} C_VEL
LIN {X 0,Y 583.614,Z 702.53,A -85,B 0,C 180,E1 1831.432,E2 1831.432} C_VEL
LIN {X 0,Y 583.736,Z 702.53,A -85,B 0,C 180,E1 1836.738,E2 1836.738} C_VEL
LIN {X 0,Y 583.746,Z 702.53,A -85,B 0,C 180,E1 1842.202,E2 1842.202} C_VEL
LIN {X 0,Y 583.534,Z 702.53,A -85,B 0,C 180,E1 1847.751,E2 1847.751} C_VEL
LIN {X 0,Y 583.523,Z 702.53,A -85,B 0,C 180,E1 1853.252,E2 1853.252} C_VEL
LIN {X 0,Y 583.733,Z 702.53,A -85,B 0,C 180,E1 1858.505,E2 1858.505} C_VEL
LIN {X 0,Y 583.636,Z 702.53,A -85,B 0,C 180,E1 1863.925,E2 1863.925} C_VEL
LIN {X 0,Y 583.652,Z 702.53,A -85,B 0,C 180,E1 1868.779,E2 1868.779} C_VEL
LIN {X 0,Y 583.772,Z 702.53,A -85,B 0,C 180,E1 1873.48,E2 1873.48} C_VEL
LIN {X 0,Y 583.859,Z 702.53,A -85,B 0,C 180,E1 1878.067,E2 1878.067} C_VEL
LIN {X 0,Y 583.933,Z 702.53,A -85,B 0,C 180,E1 1882.576,E2 1882.576} C_VEL
LIN {X 0,Y 583.992,Z 702.53,A -85,B 0,C 180,E1 1887.038,E2 1887.038} C_VEL
LIN {X 0,Y 583.795,Z 702.53,A -85,B 0,C 180,E1 1890.857,E2 1890.857} C_VEL
LIN {X 0,Y 586.646,Z 712.633,A -85,B 0,C 180,E1 1891.163,E2 1891.163} C_VEL
LIN {X 0,Y 586.672,Z 751.364,A -85,B 0,C 180,E1 1892.165,E2 1892.165} C_VEL
LIN {X 0,Y 586.152,Z 786.876,A -85,B 0,C 180,E1 1893.69,E2 1893.69} C_VEL
LIN {X 0,Y 585.576,Z 819.855,A -85,B 0,C 180,E1 1895.731,E2 1895.731} C_VEL
LIN {X 0,Y 585.105,Z 850.699,A -85,B 0,C 180,E1 1898.342,E2 1898.342} C_VEL
LIN {X 0,Y 584.693,Z 875.975,A -85,B 0,C 180,E1 1901.205,E2 1901.205} C_VEL
LIN {X 0,Y 584.373,Z 896.781,A -85,B 0,C 180,E1 1904.348,E2 1904.348} C_VEL
LIN {X 0,Y 584.265,Z 912.306,A -85,B 0,C 180,E1 1907.584,E2 1907.584} C_VEL
LIN {X 0,Y 584.181,Z 923.768,A -85,B 0,C 180,E1 1911.201,E2 1911.201} C_VEL
LIN {X 0,Y 584.03,Z 929.165,A -85,B 0,C 180,E1 1914.419,E2 1914.419} C_VEL
LIN {X 0,Y 583.989,Z 930.335,A -85,B 0,C 180,E1 1917.718,E2 1917.718} C_VEL
LIN {X 0,Y 584.099,Z 926.96,A -85,B 0,C 180,E1 1921.112,E2 1921.112} C_VEL
LIN {X 0,Y 584.258,Z 917.425,A -85,B 0,C 180,E1 1924.939,E2 1924.939} C_VEL
LIN {X 0,Y 584.266,Z 902.661,A -85,B 0,C 180,E1 1928.466,E2 1928.466} C_VEL
LIN {X 0,Y 584.539,Z 882.463,A -85,B 0,C 180,E1 1931.824,E2 1931.824} C_VEL
LIN {X 0,Y 584.931,Z 856.863,A -85,B 0,C 180,E1 1934.946,E2 1934.946} C_VEL
LIN {X 0,Y 585.45,Z 827.69,A -85,B 0,C 180,E1 1937.587,E2 1937.587} C_VEL
LIN {X 0,Y 586.03,Z 795.102,A -85,B 0,C 180,E1 1939.773,E2 1939.773} C_VEL
LIN {X 0,Y 586.595,Z 759.713,A -85,B 0,C 180,E1 1941.443,E2 1941.443} C_VEL
LIN {X 0,Y 587.008,Z 723.189,A -85,B 0,C 180,E1 1942.522,E2 1942.522} C_VEL
LIN {X 0,Y 586.29,Z 709.602,A -85,B 0,C 180,E1 1942.811,E2 1942.811} C_VEL
LIN {X 0,Y 584.058,Z 702.53,A -85,B 0,C 180,E1 1943.087,E2 1943.087} C_VEL
LIN {X 0,Y 583.655,Z 702.53,A -85,B 0,C 180,E1 1948.885,E2 1948.885} C_VEL
LIN {X 0,Y 583.808,Z 702.53,A -85,B 0,C 180,E1 1954.781,E2 1954.781} C_VEL
LIN {X 0,Y 583.931,Z 702.53,A -85,B 0,C 180,E1 1960.387,E2 1960.387} C_VEL
LIN {X 0,Y 584.118,Z 702.53,A -85,B 0,C 180,E1 1966.571,E2 1966.571} C_VEL
LIN {X 0,Y 583.876,Z 702.53,A -85,B 0,C 180,E1 1972.7,E2 1972.7} C_VEL
LIN {X 0,Y 584.019,Z 702.53,A -85,B 0,C 180,E1 1977.05,E2 1977.05} C_VEL
LIN {X 0,Y 583.905,Z 702.53,A -85,B 0,C 180,E1 1982.444,E2 1982.444} C_VEL
LIN {X 0,Y 584.077,Z 702.53,A -85,B 0,C 180,E1 1985.794,E2 1985.794} C_VEL
LIN {X 0,Y 581.614,Z 702.53,A -85,B 0,C 180,E1 1987.055,E2 1987.055} C_VEL
LIN {X 0,Y 575.952,Z 702.53,A -85,B 0,C 180,E1 1988.94,E2 1988.94} C_VEL
LIN {X 0,Y 575.849,Z 702.53,A -85,B 0,C 180,E1 1989.159,E2 1989.159} C_VEL
LIN {X 0,Y 575.911,Z 702.53,A -85,B 0,C 180,E1 1995.199,E2 1995.199} C_VEL
LIN {X 0,Y 575.804,Z 702.53,A -85,B 0,C 180,E1 2001.532,E2 2001.532} C_VEL
LIN {X 0,Y 575.695,Z 702.53,A -85,B 0,C 180,E1 2006.973,E2 2006.973} C_VEL
LIN {X 0,Y 575.655,Z 702.53,A -85,B 0,C 180,E1 2011.626,E2 2011.626} C_VEL
LIN {X 0,Y 575.833,Z 702.53,A -85,B 0,C 180,E1 2017.071,E2 2017.071} C_VEL
LIN {X 0,Y 575.797,Z 702.53,A -85,B 0,C 180,E1 2022.957,E2 2022.957} C_VEL
LIN {X 0,Y 575.679,Z 702.53,A -85,B 0,C 180,E1 2029.482,E2 2029.482} C_VEL
LIN {X 0,Y 575.713,Z 702.53,A -85,B 0,C 180,E1 2034.784,E2 2034.784} C_VEL
LIN {X 0,Y 576.017,Z 702.53,A -85,B 0,C 180,E1 2038.578,E2 2038.578} C_VEL
LIN {X 0,Y 580.959,Z 716.932,A -85,B 0,C 180,E1 2039.098,E2 2039.098} C_VEL
LIN {X 0,Y 580.834,Z 777.583,A -85,B 0,C 180,E1 2040.094,E2 2040.094} C_VEL
LIN {X 0,Y 580.278,Z 816.581,A -85,B 0,C 180,E1 2041.355,E2 2041.355} C_VEL
LIN {X 0,Y 579.445,Z 853.619,A -85,B 0,C 180,E1 2043.167,E2 2043.167} C_VEL
LIN {X 0,Y 578.483,Z 889.85,A -85,B 0,C 180,E1 2045.633,E2 2045.633} C_VEL
LIN {X 0,Y 577.683,Z 920.633,A -85,B 0,C 180,E1 2048.41,E2 2048.41} C_VEL
LIN {X 0,Y 577.015,Z 948.701,A -85,B 0,C 180,E1 2051.71,E2 2051.71} C_VEL
LIN {X 0,Y 576.559,Z 971.561,A -85,B 0,C 180,E1 2055.253,E2 2055.253} C_VEL
LIN {X 0,Y 576.342,Z 989.852,A -85,B 0,C 180,E1 2059.141,E2 2059.141} C_VEL
LIN {X 0,Y 576.221,Z 1000.677,A -85,B 0,C 180,E1 2062.476,E2 2062.476} C_VEL
LIN {X 0,Y 576.085,Z 1006.956,A -85,B 0,C 180,E1 2065.493,E2 2065.493} C_VEL
LIN {X 0,Y 576.128,Z 1010.086,A -85,B 0,C 180,E1 2068.499,E2 2068.499} C_VEL
LIN {X 0,Y 576.277,Z 1010.087,A -85,B 0,C 180,E1 2071.5,E2 2071.5} C_VEL
LIN {X 0,Y 576.257,Z 1004.878,A -85,B 0,C 180,E1 2075.694,E2 2075.694} C_VEL
LIN {X 0,Y 576.291,Z 995.073,A -85,B 0,C 180,E1 2079.419,E2 2079.419} C_VEL
LIN {X 0,Y 576.455,Z 979.448,A -85,B 0,C 180,E1 2083.241,E2 2083.241} C_VEL
LIN {X 0,Y 576.774,Z 958.401,A -85,B 0,C 180,E1 2086.914,E2 2086.914} C_VEL
LIN {X 0,Y 577.38,Z 932.869,A -85,B 0,C 180,E1 2090.261,E2 2090.261} C_VEL
LIN {X 0,Y 578.127,Z 902.629,A -85,B 0,C 180,E1 2093.301,E2 2093.301} C_VEL
LIN {X 0,Y 579.021,Z 868.727,A -85,B 0,C 180,E1 2095.894,E2 2095.894} C_VEL
LIN {X 0,Y 579.921,Z 832.751,A -85,B 0,C 180,E1 2097.929,E2 2097.929} C_VEL
LIN {X 0,Y 580.61,Z 795.492,A -85,B 0,C 180,E1 2099.399,E2 2099.399} C_VEL
LIN {X 0,Y 581.114,Z 758.885,A -85,B 0,C 180,E1 2100.281,E2 2100.281} C_VEL
LIN {X 0,Y 580.312,Z 713.538,A -85,B 0,C 180,E1 2100.989,E2 2100.989} C_VEL
LIN {X 0,Y 575.801,Z 702.53,A -85,B 0,C 180,E1 2101.497,E2 2101.497} C_VEL
LIN {X 0,Y 575.823,Z 702.53,A -85,B 0,C 180,E1 2107.067,E2 2107.067} C_VEL
LIN {X 0,Y 575.81,Z 702.53,A -85,B 0,C 180,E1 2112.951,E2 2112.951} C_VEL
LIN {X 0,Y 575.644,Z 702.53,A -85,B 0,C 180,E1 2119.049,E2 2119.049} C_VEL
LIN {X 0,Y 575.704,Z 702.53,A -85,B 0,C 180,E1 2124.779,E2 2124.779} C_VEL
LIN {X 0,Y 575.807,Z 702.53,A -85,B 0,C 180,E1 2130.13,E2 2130.13} C_VEL
LIN {X 0,Y 575.752,Z 702.53,A -85,B 0,C 180,E1 2135.199,E2 2135.199} C_VEL
LIN {X 0,Y 575.81,Z 702.53,A -85,B 0,C 180,E1 2140.639,E2 2140.639} C_VEL
LIN {X 0,Y 576.03,Z 702.53,A -85,B 0,C 180,E1 2146.354,E2 2146.354} C_VEL
LIN {X 0,Y 576.021,Z 702.53,A -85,B 0,C 180,E1 2152.463,E2 2152.463} C_VEL
LIN {X 0,Y 576.141,Z 702.53,A -85,B 0,C 180,E1 2156.986,E2 2156.986} C_VEL
LIN {X 0,Y 576.247,Z 702.53,A -85,B 0,C 180,E1 2161.488,E2 2161.488} C_VEL
LIN {X 0,Y 576.237,Z 702.53,A -85,B 0,C 180,E1 2165.999,E2 2165.999} C_VEL
LIN {X 0,Y 575.874,Z 702.53,A -85,B 0,C 180,E1 2172.086,E2 2172.086} C_VEL
LIN {X 0,Y 575.887,Z 702.53,A -85,B 0,C 180,E1 2176.736,E2 2176.736} C_VEL
LIN {X 0,Y 575.833,Z 702.53,A -85,B 0,C 180,E1 2181.505,E2 2181.505} C_VEL
LIN {X 0,Y 575.673,Z 702.53,A -85,B 0,C 180,E1 2186.97,E2 2186.97} C_VEL
LIN {X 0,Y 575.706,Z 702.53,A -85,B 0,C 180,E1 2191.594,E2 2191.594} C_VEL
LIN {X 0,Y 575.82,Z 702.53,A -85,B 0,C 180,E1 2197.042,E2 2197.042} C_VEL
LIN {X 0,Y 575.825,Z 702.53,A -85,B 0,C 180,E1 2202.921,E2 2202.921} C_VEL
LIN {X 0,Y 575.688,Z 702.53,A -85,B 0,C 180,E1 2209.444,E2 2209.444} C_VEL
LIN {X 0,Y 575.672,Z 702.53,A -85,B 0,C 180,E1 2214.782,E2 2214.782} C_VEL
LIN {X 0,Y 575.803,Z 702.53,A -85,B 0,C 180,E1 2220.136,E2 2220.136} C_VEL
LIN {X 0,Y 575.808,Z 702.53,A -85,B 0,C 180,E1 2226.465,E2 2226.465} C_VEL
LIN {X 0,Y 575.933,Z 702.53,A -85,B 0,C 180,E1 2231.675,E2 2231.675} C_VEL
LIN {X 0,Y 575.955,Z 702.53,A -85,B 0,C 180,E1 2237.901,E2 2237.901} C_VEL
LIN {X 0,Y 576.028,Z 702.53,A -85,B 0,C 180,E1 2242.474,E2 2242.474} C_VEL
LIN {X 0,Y 576.087,Z 702.53,A -85,B 0,C 180,E1 2246.997,E2 2246.997} C_VEL
LIN {X 0,Y 575.812,Z 702.53,A -85,B 0,C 180,E1 2250.469,E2 2250.469} C_VEL
LIN {X 0,Y 579.578,Z 716.094,A -85,B 0,C 180,E1 2250.886,E2 2250.886} C_VEL
LIN {X 0,Y 579.411,Z 753.514,A -85,B 0,C 180,E1 2251.912,E2 2251.912} C_VEL
LIN {X 0,Y 578.761,Z 788.382,A -85,B 0,C 180,E1 2253.457,E2 2253.457} C_VEL
LIN {X 0,Y 578.021,Z 822.294,A -85,B 0,C 180,E1 2255.618,E2 2255.618} C_VEL
LIN {X 0,Y 577.404,Z 852.448,A -85,B 0,C 180,E1 2258.265,E2 2258.265} C_VEL
LIN {X 0,Y 576.916,Z 878.758,A -85,B 0,C 180,E1 2261.358,E2 2261.358} C_VEL
LIN {X 0,Y 576.526,Z 900.122,A -85,B 0,C 180,E1 2264.79,E2 2264.79} C_VEL
LIN {X 0,Y 576.35,Z 915.495,A -85,B 0,C 180,E1 2268.312,E2 2268.312} C_VEL
LIN {X 0,Y 576.194,Z 925.493,A -85,B 0,C 180,E1 2271.941,E2 2271.941} C_VEL
LIN {X 0,Y 576.117,Z 929.556,A -85,B 0,C 180,E1 2274.777,E2 2274.777} C_VEL
LIN {X 0,Y 576.088,Z 930.226,A -85,B 0,C 180,E1 2278.132,E2 2278.132} C_VEL
LIN {X 0,Y 576.203,Z 926.277,A -85,B 0,C 180,E1 2281.587,E2 2281.587} C_VEL
LIN {X 0,Y 576.323,Z 916.992,A -85,B 0,C 180,E1 2285.173,E2 2285.173} C_VEL
LIN {X 0,Y 576.422,Z 902.92,A -85,B 0,C 180,E1 2288.574,E2 2288.574} C_VEL
LIN {X 0,Y 576.728,Z 883.728,A -85,B 0,C 180,E1 2291.846,E2 2291.846} C_VEL
LIN {X 0,Y 577.224,Z 858.247,A -85,B 0,C 180,E1 2295.046,E2 2295.046} C_VEL
LIN {X 0,Y 577.904,Z 828.89,A -85,B 0,C 180,E1 2297.773,E2 2297.773} C_VEL
LIN {X 0,Y 578.621,Z 796.276,A -85,B 0,C 180,E1 2300.012,E2 2300.012} C_VEL
LIN {X 0,Y 579.338,Z 760.921,A -85,B 0,C 180,E1 2301.724,E2 2301.724} C_VEL
LIN {X 0,Y 579.883,Z 723.6,A -85,B 0,C 180,E1 2302.851,E2 2302.851} C_VEL
LIN {X 0,Y 579.153,Z 711.648,A -85,B 0,C 180,E1 2303.121,E2 2303.121} C_VEL
LIN {X 0,Y 576.064,Z 702.53,A -85,B 0,C 180,E1 2303.512,E2 2303.512} C_VEL
LIN {X 0,Y 575.727,Z 702.53,A -85,B 0,C 180,E1 2310.154,E2 2310.154} C_VEL
LIN {X 0,Y 575.854,Z 702.53,A -85,B 0,C 180,E1 2315.23,E2 2315.23} C_VEL
LIN {X 0,Y 576.026,Z 702.53,A -85,B 0,C 180,E1 2320.579,E2 2320.579} C_VEL
LIN {X 0,Y 576.169,Z 702.53,A -85,B 0,C 180,E1 2326.382,E2 2326.382} C_VEL
LIN {X 0,Y 575.955,Z 702.53,A -85,B 0,C 180,E1 2332.687,E2 2332.687} C_VEL
LIN {X 0,Y 576.111,Z 702.53,A -85,B 0,C 180,E1 2337.01,E2 2337.01} C_VEL
LIN {X 0,Y 576.256,Z 702.53,A -85,B 0,C 180,E1 2341.512,E2 2341.512} C_VEL
LIN {X 0,Y 576.189,Z 702.53,A -85,B 0,C 180,E1 2346.024,E2 2346.024} C_VEL
LIN {X 0,Y 575.849,Z 702.53,A -85,B 0,C 180,E1 2349.159,E2 2349.159} C_VEL
LIN {X 0,Y 571.91,Z 702.53,A -85,B 0,C 180,E1 2350.858,E2 2350.858} C_VEL
LIN {X 0,Y 567.89,Z 702.53,A -85,B 0,C 180,E1 2352.581,E2 2352.581} C_VEL
LIN {X 0,Y 567.918,Z 702.53,A -85,B 0,C 180,E1 2357.003,E2 2357.003} C_VEL
LIN {X 0,Y 567.875,Z 702.53,A -85,B 0,C 180,E1 2361.848,E2 2361.848} C_VEL
LIN {X 0,Y 567.805,Z 702.53,A -85,B 0,C 180,E1 2366.866,E2 2366.866} C_VEL
LIN {X 0,Y 567.687,Z 702.53,A -85,B 0,C 180,E1 2372.122,E2 2372.122} C_VEL
LIN {X 0,Y 567.905,Z 702.53,A -85,B 0,C 180,E1 2377.678,E2 2377.678} C_VEL
LIN {X 0,Y 567.786,Z 702.53,A -85,B 0,C 180,E1 2383.714,E2 2383.714} C_VEL
LIN {X 0,Y 567.67,Z 702.53,A -85,B 0,C 180,E1 2388.35,E2 2388.35} C_VEL
LIN {X 0,Y 567.738,Z 702.53,A -85,B 0,C 180,E1 2394.214,E2 2394.214} C_VEL
LIN {X 0,Y 568.092,Z 702.53,A -85,B 0,C 180,E1 2398.088,E2 2398.088} C_VEL
LIN {X 0,Y 574.173,Z 717.31,A -85,B 0,C 180,E1 2398.697,E2 2398.697} C_VEL
LIN {X 0,Y 573.973,Z 777.582,A -85,B 0,C 180,E1 2399.699,E2 2399.699} C_VEL
LIN {X 0,Y 573.251,Z 816.801,A -85,B 0,C 180,E1 2400.98,E2 2400.98} C_VEL
LIN {X 0,Y 572.257,Z 853.79,A -85,B 0,C 180,E1 2402.813,E2 2402.813} C_VEL
LIN {X 0,Y 571.09,Z 889.843,A -85,B 0,C 180,E1 2405.296,E2 2405.296} C_VEL
LIN {X 0,Y 570.115,Z 920.907,A -85,B 0,C 180,E1 2408.138,E2 2408.138} C_VEL
LIN {X 0,Y 569.312,Z 948.702,A -85,B 0,C 180,E1 2411.453,E2 2411.453} C_VEL
LIN {X 0,Y 568.755,Z 971.201,A -85,B 0,C 180,E1 2414.981,E2 2414.981} C_VEL
LIN {X 0,Y 568.414,Z 987.982,A -85,B 0,C 180,E1 2418.516,E2 2418.516} C_VEL
LIN {X 0,Y 568.321,Z 1000.677,A -85,B 0,C 180,E1 2422.371,E2 2422.371} C_VEL
LIN {X 0,Y 568.206,Z 1006.956,A -85,B 0,C 180,E1 2425.43,E2 2425.43} C_VEL
LIN {X 0,Y 568.258,Z 1010.086,A -85,B 0,C 180,E1 2428.478,E2 2428.478} C_VEL
LIN {X 0,Y 568.393,Z 1010.087,A -85,B 0,C 180,E1 2431.521,E2 2431.521} C_VEL
LIN {X 0,Y 568.365,Z 1005.389,A -85,B 0,C 180,E1 2435.522,E2 2435.522} C_VEL
LIN {X 0,Y 568.38,Z 995.072,A -85,B 0,C 180,E1 2439.551,E2 2439.551} C_VEL
LIN {X 0,Y 568.6,Z 979.447,A -85,B 0,C 180,E1 2443.428,E2 2443.428} C_VEL
LIN {X 0,Y 569.048,Z 958.159,A -85,B 0,C 180,E1 2447.187,E2 2447.187} C_VEL
LIN {X 0,Y 569.73,Z 932.868,A -85,B 0,C 180,E1 2450.545,E2 2450.545} C_VEL
LIN {X 0,Y 570.648,Z 903.125,A -85,B 0,C 180,E1 2453.58,E2 2453.58} C_VEL
LIN {X 0,Y 571.712,Z 869.76,A -85,B 0,C 180,E1 2456.179,E2 2456.179} C_VEL
LIN {X 0,Y 572.802,Z 834.438,A -85,B 0,C 180,E1 2458.222,E2 2458.222} C_VEL
LIN {X 0,Y 573.637,Z 798.386,A -85,B 0,C 180,E1 2459.695,E2 2459.695} C_VEL
LIN {X 0,Y 574.287,Z 762.522,A -85,B 0,C 180,E1 2460.618,E2 2460.618} C_VEL
LIN {X 0,Y 573.659,Z 716.027,A -85,B 0,C 180,E1 2461.353,E2 2461.353} C_VEL
LIN {X 0,Y 567.841,Z 702.53,A -85,B 0,C 180,E1 2461.955,E2 2461.955} C_VEL
LIN {X 0,Y 567.894,Z 702.53,A -85,B 0,C 180,E1 2467.673,E2 2467.673} C_VEL
LIN {X 0,Y 567.806,Z 702.53,A -85,B 0,C 180,E1 2473.708,E2 2473.708} C_VEL
LIN {X 0,Y 567.68,Z 702.53,A -85,B 0,C 180,E1 2478.347,E2 2478.347} C_VEL
LIN {X 0,Y 567.731,Z 702.53,A -85,B 0,C 180,E1 2484.209,E2 2484.209} C_VEL
LIN {X 0,Y 567.9,Z 702.53,A -85,B 0,C 180,E1 2489.671,E2 2489.671} C_VEL
LIN {X 0,Y 567.797,Z 702.53,A -85,B 0,C 180,E1 2494.828,E2 2494.828} C_VEL
LIN {X 0,Y 567.83,Z 702.53,A -85,B 0,C 180,E1 2499.781,E2 2499.781} C_VEL
LIN {X 0,Y 567.912,Z 702.53,A -85,B 0,C 180,E1 2504.582,E2 2504.582} C_VEL
LIN {X 0,Y 567.943,Z 702.53,A -85,B 0,C 180,E1 2509.447,E2 2509.447} C_VEL
LIN {X 0,Y 567.999,Z 702.53,A -85,B 0,C 180,E1 2513.889,E2 2513.889} C_VEL
LIN {X 0,Y 567.989,Z 702.53,A -85,B 0,C 180,E1 2518.466,E2 2518.466} C_VEL
LIN {X 0,Y 568.048,Z 702.53,A -85,B 0,C 180,E1 2523.033,E2 2523.033} C_VEL
LIN {X 0,Y 567.976,Z 702.53,A -85,B 0,C 180,E1 2527.62,E2 2527.62} C_VEL
LIN {X 0,Y 567.959,Z 702.53,A -85,B 0,C 180,E1 2532.257,E2 2532.257} C_VEL
LIN {X 0,Y 567.957,Z 702.53,A -85,B 0,C 180,E1 2536.977,E2 2536.977} C_VEL
LIN {X 0,Y 567.873,Z 702.53,A -85,B 0,C 180,E1 2541.822,E2 2541.822} C_VEL
LIN {X 0,Y 567.789,Z 702.53,A -85,B 0,C 180,E1 2546.839,E2 2546.839} C_VEL
LIN {X 0,Y 567.77,Z 702.53,A -85,B 0,C 180,E1 2552.088,E2 2552.088} C_VEL
LIN {X 0,Y 567.887,Z 702.53,A -85,B 0,C 180,E1 2557.648,E2 2557.648} C_VEL
LIN {X 0,Y 567.821,Z 702.53,A -85,B 0,C 180,E1 2563.677,E2 2563.677} C_VEL
LIN {X 0,Y 567.681,Z 702.53,A -85,B 0,C 180,E1 2568.352,E2 2568.352} C_VEL
LIN {X 0,Y 567.708,Z 702.53,A -85,B 0,C 180,E1 2574.213,E2 2574.213} C_VEL
LIN {X 0,Y 567.909,Z 702.53,A -85,B 0,C 180,E1 2579.678,E2 2579.678} C_VEL
LIN {X 0,Y 567.822,Z 702.53,A -85,B 0,C 180,E1 2584.836,E2 2584.836} C_VEL
LIN {X 0,Y 567.874,Z 702.53,A -85,B 0,C 180,E1 2589.791,E2 2589.791} C_VEL
LIN {X 0,Y 567.893,Z 702.53,A -85,B 0,C 180,E1 2594.59,E2 2594.59} C_VEL
LIN {X 0,Y 567.96,Z 702.53,A -85,B 0,C 180,E1 2599.3,E2 2599.3} C_VEL
LIN {X 0,Y 568.002,Z 702.53,A -85,B 0,C 180,E1 2603.9,E2 2603.9} C_VEL
LIN {X 0,Y 567.825,Z 702.53,A -85,B 0,C 180,E1 2608.477,E2 2608.477} C_VEL
LIN {X 0,Y 567.858,Z 702.53,A -85,B 0,C 180,E1 2610.048,E2 2610.048} C_VEL
LIN {X 0,Y 572.474,Z 717.442,A -85,B 0,C 180,E1 2610.567,E2 2610.567} C_VEL
LIN {X 0,Y 572.201,Z 754.346,A -85,B 0,C 180,E1 2611.606,E2 2611.606} C_VEL
LIN {X 0,Y 571.393,Z 789.875,A -85,B 0,C 180,E1 2613.217,E2 2613.217} C_VEL
LIN {X 0,Y 570.484,Z 823.381,A -85,B 0,C 180,E1 2615.407,E2 2615.407} C_VEL
LIN {X 0,Y 569.767,Z 852.335,A -85,B 0,C 180,E1 2617.993,E2 2617.993} C_VEL
LIN {X 0,Y 569.141,Z 878.594,A -85,B 0,C 180,E1 2621.118,E2 2621.118} C_VEL
LIN {X 0,Y 568.688,Z 899.558,A -85,B 0,C 180,E1 2624.507,E2 2624.507} C_VEL
LIN {X 0,Y 568.484,Z 915.564,A -85,B 0,C 180,E1 2628.212,E2 2628.212} C_VEL
LIN {X 0,Y 568.336,Z 925.394,A -85,B 0,C 180,E1 2631.822,E2 2631.822} C_VEL
LIN {X 0,Y 568.161,Z 930.054,A -85,B 0,C 180,E1 2635.497,E2 2635.497} C_VEL
LIN {X 0,Y 568.166,Z 929.777,A -85,B 0,C 180,E1 2638.831,E2 2638.831} C_VEL
LIN {X 0,Y 568.305,Z 925.416,A -85,B 0,C 180,E1 2642.077,E2 2642.077} C_VEL
LIN {X 0,Y 568.387,Z 915.431,A -85,B 0,C 180,E1 2645.739,E2 2645.739} C_VEL
LIN {X 0,Y 568.587,Z 900.408,A -85,B 0,C 180,E1 2649.236,E2 2649.236} C_VEL
LIN {X 0,Y 569.017,Z 880.088,A -85,B 0,C 180,E1 2652.591,E2 2652.591} C_VEL
LIN {X 0,Y 569.651,Z 854.79,A -85,B 0,C 180,E1 2655.663,E2 2655.663} C_VEL
LIN {X 0,Y 570.478,Z 825.12,A -85,B 0,C 180,E1 2658.363,E2 2658.363} C_VEL
LIN {X 0,Y 571.368,Z 791.385,A -85,B 0,C 180,E1 2660.61,E2 2660.61} C_VEL
LIN {X 0,Y 572.191,Z 756.106,A -85,B 0,C 180,E1 2662.238,E2 2662.238} C_VEL
LIN {X 0,Y 572.834,Z 720.958,A -85,B 0,C 180,E1 2663.25,E2 2663.25} C_VEL
LIN {X 0,Y 571.463,Z 712.195,A -85,B 0,C 180,E1 2663.492,E2 2663.492} C_VEL
LIN {X 0,Y 568.075,Z 702.53,A -85,B 0,C 180,E1 2663.884,E2 2663.884} C_VEL
LIN {X 0,Y 567.84,Z 702.53,A -85,B 0,C 180,E1 2669.696,E2 2669.696} C_VEL
LIN {X 0,Y 567.904,Z 702.53,A -85,B 0,C 180,E1 2674.86,E2 2674.86} C_VEL
LIN {X 0,Y 568.04,Z 702.53,A -85,B 0,C 180,E1 2679.815,E2 2679.815} C_VEL
LIN {X 0,Y 568.244,Z 702.53,A -85,B 0,C 180,E1 2686.188,E2 2686.188} C_VEL
LIN {X 0,Y 568.031,Z 702.53,A -85,B 0,C 180,E1 2692.675,E2 2692.675} C_VEL
LIN {X 0,Y 568.206,Z 702.53,A -85,B 0,C 180,E1 2696.968,E2 2696.968} C_VEL
LIN {X 0,Y 568.369,Z 702.53,A -85,B 0,C 180,E1 2701.533,E2 2701.533} C_VEL
LIN {X 0,Y 568.257,Z 702.53,A -85,B 0,C 180,E1 2706.108,E2 2706.108} C_VEL
LIN {X 0,Y 567.927,Z 702.53,A -85,B 0,C 180,E1 2712.282,E2 2712.282} C_VEL
LIN {X 0,Y 567.89,Z 702.53,A -85,B 0,C 180,E1 2712.581,E2 2712.581} C_VEL
LIN {X 0,Y 563.951,Z 702.53,A -85,B 0,C 180,E1 2714.302,E2 2714.302} C_VEL
LIN {X 0,Y 559.987,Z 702.53,A -85,B 0,C 180,E1 2716.047,E2 2716.047} C_VEL
LIN {X 0,Y 559.925,Z 702.53,A -85,B 0,C 180,E1 2722.175,E2 2722.175} C_VEL
LIN {X 0,Y 559.852,Z 702.53,A -85,B 0,C 180,E1 2727.279,E2 2727.279} C_VEL
LIN {X 0,Y 559.715,Z 702.53,A -85,B 0,C 180,E1 2732.636,E2 2732.636} C_VEL
LIN {X 0,Y 559.904,Z 702.53,A -85,B 0,C 180,E1 2738.313,E2 2738.313} C_VEL
LIN {X 0,Y 559.812,Z 702.53,A -85,B 0,C 180,E1 2744.5,E2 2744.5} C_VEL
LIN {X 0,Y 559.738,Z 702.53,A -85,B 0,C 180,E1 2749.682,E2 2749.682} C_VEL
LIN {X 0,Y 559.957,Z 702.53,A -85,B 0,C 180,E1 2755.533,E2 2755.533} C_VEL
LIN {X 0,Y 560.143,Z 703.258,A -85,B 0,C 180,E1 2757.611,E2 2757.611} C_VEL
LIN {X 0,Y 567.409,Z 720.438,A -85,B 0,C 180,E1 2758.326,E2 2758.326} C_VEL
LIN {X 0,Y 567.133,Z 777.601,A -85,B 0,C 180,E1 2759.295,E2 2759.295} C_VEL
LIN {X 0,Y 566.331,Z 816.291,A -85,B 0,C 180,E1 2760.568,E2 2760.568} C_VEL
LIN {X 0,Y 565.092,Z 853.707,A -85,B 0,C 180,E1 2762.434,E2 2762.434} C_VEL
LIN {X 0,Y 563.759,Z 889.561,A -85,B 0,C 180,E1 2764.929,E2 2764.929} C_VEL
LIN {X 0,Y 562.576,Z 920.125,A -85,B 0,C 180,E1 2767.745,E2 2767.745} C_VEL
LIN {X 0,Y 561.599,Z 947.676,A -85,B 0,C 180,E1 2771.046,E2 2771.046} C_VEL
LIN {X 0,Y 560.925,Z 969.168,A -85,B 0,C 180,E1 2774.394,E2 2774.394} C_VEL
LIN {X 0,Y 560.564,Z 986.441,A -85,B 0,C 180,E1 2777.958,E2 2777.958} C_VEL
LIN {X 0,Y 560.461,Z 999.717,A -85,B 0,C 180,E1 2781.874,E2 2781.874} C_VEL
LIN {X 0,Y 560.335,Z 1006.956,A -85,B 0,C 180,E1 2785.366,E2 2785.366} C_VEL
LIN {X 0,Y 560.357,Z 1010.087,A -85,B 0,C 180,E1 2788.457,E2 2788.457} C_VEL
LIN {X 0,Y 560.487,Z 1010.087,A -85,B 0,C 180,E1 2791.543,E2 2791.543} C_VEL
LIN {X 0,Y 560.468,Z 1005.838,A -85,B 0,C 180,E1 2795.356,E2 2795.356} C_VEL
LIN {X 0,Y 560.524,Z 996.303,A -85,B 0,C 180,E1 2799.296,E2 2799.296} C_VEL
LIN {X 0,Y 560.772,Z 981.281,A -85,B 0,C 180,E1 2803.222,E2 2803.222} C_VEL
LIN {X 0,Y 561.22,Z 960.919,A -85,B 0,C 180,E1 2807.002,E2 2807.002} C_VEL
LIN {X 0,Y 562.065,Z 934.614,A -85,B 0,C 180,E1 2810.633,E2 2810.633} C_VEL
LIN {X 0,Y 563.197,Z 903.996,A -85,B 0,C 180,E1 2813.831,E2 2813.831} C_VEL
LIN {X 0,Y 564.4,Z 871.198,A -85,B 0,C 180,E1 2816.443,E2 2816.443} C_VEL
LIN {X 0,Y 565.688,Z 836.236,A -85,B 0,C 180,E1 2818.517,E2 2818.517} C_VEL
LIN {X 0,Y 566.702,Z 799.486,A -85,B 0,C 180,E1 2820.059,E2 2820.059} C_VEL
LIN {X 0,Y 567.485,Z 763.308,A -85,B 0,C 180,E1 2821.011,E2 2821.011} C_VEL
LIN {X 0,Y 567.081,Z 719.099,A -85,B 0,C 180,E1 2821.714,E2 2821.714} C_VEL
LIN {X 0,Y 559.837,Z 702.53,A -85,B 0,C 180,E1 2822.454,E2 2822.454} C_VEL
LIN {X 0,Y 559.895,Z 702.53,A -85,B 0,C 180,E1 2828.308,E2 2828.308} C_VEL
LIN {X 0,Y 559.839,Z 702.53,A -85,B 0,C 180,E1 2834.493,E2 2834.493} C_VEL
LIN {X 0,Y 559.739,Z 702.53,A -85,B 0,C 180,E1 2839.677,E2 2839.677} C_VEL
LIN {X 0,Y 559.937,Z 702.53,A -85,B 0,C 180,E1 2845.526,E2 2845.526} C_VEL
LIN {X 0,Y 559.95,Z 702.53,A -85,B 0,C 180,E1 2850.975,E2 2850.975} C_VEL
LIN {X 0,Y 559.956,Z 702.53,A -85,B 0,C 180,E1 2856.386,E2 2856.386} C_VEL
LIN {X 0,Y 560.099,Z 702.53,A -85,B 0,C 180,E1 2862.752,E2 2862.752} C_VEL
LIN {X 0,Y 560.156,Z 702.53,A -85,B 0,C 180,E1 2867.545,E2 2867.545} C_VEL
LIN {X 0,Y 560.228,Z 702.53,A -85,B 0,C 180,E1 2872.249,E2 2872.249} C_VEL
LIN {X 0,Y 560.324,Z 702.53,A -85,B 0,C 180,E1 2876.901,E2 2876.901} C_VEL
LIN {X 0,Y 560.451,Z 702.53,A -85,B 0,C 180,E1 2881.53,E2 2881.53} C_VEL
LIN {X 0,Y 560.382,Z 702.53,A -85,B 0,C 180,E1 2886.17,E2 2886.17} C_VEL
LIN {X 0,Y 560.038,Z 702.53,A -85,B 0,C 180,E1 2892.433,E2 2892.433} C_VEL
LIN {X 0,Y 560.021,Z 702.53,A -85,B 0,C 180,E1 2897.225,E2 2897.225} C_VEL
LIN {X 0,Y 559.922,Z 702.53,A -85,B 0,C 180,E1 2902.148,E2 2902.148} C_VEL
LIN {X 0,Y 559.828,Z 702.53,A -85,B 0,C 180,E1 2907.252,E2 2907.252} C_VEL
LIN {X 0,Y 559.788,Z 702.53,A -85,B 0,C 180,E1 2912.602,E2 2912.602} C_VEL
LIN {X 0,Y 559.9,Z 702.53,A -85,B 0,C 180,E1 2918.281,E2 2918.281} C_VEL
LIN {X 0,Y 559.881,Z 702.53,A -85,B 0,C 180,E1 2923.305,E2 2923.305} C_VEL
LIN {X 0,Y 559.759,Z 702.53,A -85,B 0,C 180,E1 2928.977,E2 2928.977} C_VEL
LIN {X 0,Y 559.812,Z 702.53,A -85,B 0,C 180,E1 2933.927,E2 2933.927} C_VEL
LIN {X 0,Y 560.014,Z 702.53,A -85,B 0,C 180,E1 2939.526,E2 2939.526} C_VEL
LIN {X 0,Y 559.898,Z 702.53,A -85,B 0,C 180,E1 2944.455,E2 2944.455} C_VEL
LIN {X 0,Y 559.977,Z 702.53,A -85,B 0,C 180,E1 2950.517,E2 2950.517} C_VEL
LIN {X 0,Y 560.146,Z 702.53,A -85,B 0,C 180,E1 2955.968,E2 2955.968} C_VEL
LIN {X 0,Y 560.211,Z 702.53,A -85,B 0,C 180,E1 2962.26,E2 2962.26} C_VEL
LIN {X 0,Y 560.275,Z 702.53,A -85,B 0,C 180,E1 2966.912,E2 2966.912} C_VEL
LIN {X 0,Y 559.925,Z 702.53,A -85,B 0,C 180,E1 2969.662,E2 2969.662} C_VEL
LIN {X 0,Y 565.413,Z 718.732,A -85,B 0,C 180,E1 2970.239,E2 2970.239} C_VEL
LIN {X 0,Y 564.995,Z 755.195,A -85,B 0,C 180,E1 2971.291,E2 2971.291} C_VEL
LIN {X 0,Y 564.083,Z 789.61,A -85,B 0,C 180,E1 2972.875,E2 2972.875} C_VEL
LIN {X 0,Y 562.999,Z 823.228,A -85,B 0,C 180,E1 2975.094,E2 2975.094} C_VEL
LIN {X 0,Y 562.141,Z 852.222,A -85,B 0,C 180,E1 2977.714,E2 2977.714} C_VEL
LIN {X 0,Y 561.39,Z 878.248,A -85,B 0,C 180,E1 2980.846,E2 2980.846} C_VEL
LIN {X 0,Y 560.838,Z 899.729,A -85,B 0,C 180,E1 2984.364,E2 2984.364} C_VEL
LIN {X 0,Y 560.613,Z 915.374,A -85,B 0,C 180,E1 2988.032,E2 2988.032} C_VEL
LIN {X 0,Y 560.49,Z 924.359,A -85,B 0,C 180,E1 2991.233,E2 2991.233} C_VEL
LIN {X 0,Y 560.296,Z 928.638,A -85,B 0,C 180,E1 2993.828,E2 2993.828} C_VEL
LIN {X 0,Y 560.228,Z 930.427,A -85,B 0,C 180,E1 2997.32,E2 2997.32} C_VEL
LIN {X 0,Y 560.424,Z 927.758,A -85,B 0,C 180,E1 3000.771,E2 3000.771} C_VEL
LIN {X 0,Y 560.568,Z 919.964,A -85,B 0,C 180,E1 3004.424,E2 3004.424} C_VEL
LIN {X 0,Y 560.733,Z 907.909,A -85,B 0,C 180,E1 3007.808,E2 3007.808} C_VEL
LIN {X 0,Y 561.095,Z 889.315,A -85,B 0,C 180,E1 3011.392,E2 3011.392} C_VEL
LIN {X 0,Y 561.717,Z 865.614,A -85,B 0,C 180,E1 3014.708,E2 3014.708} C_VEL
LIN {X 0,Y 562.601,Z 837.569,A -85,B 0,C 180,E1 3017.61,E2 3017.61} C_VEL
LIN {X 0,Y 563.562,Z 806.078,A -85,B 0,C 180,E1 3020.039,E2 3020.039} C_VEL
LIN {X 0,Y 564.638,Z 770.419,A -85,B 0,C 180,E1 3021.998,E2 3021.998} C_VEL
LIN {X 0,Y 565.485,Z 734.948,A -85,B 0,C 180,E1 3023.269,E2 3023.269} C_VEL
LIN {X 0,Y 564.864,Z 715.51,A -85,B 0,C 180,E1 3023.769,E2 3023.769} C_VEL
LIN {X 0,Y 560.095,Z 702.53,A -85,B 0,C 180,E1 3024.308,E2 3024.308} C_VEL
LIN {X 0,Y 559.885,Z 702.53,A -85,B 0,C 180,E1 3031,E2 3031} C_VEL
LIN {X 0,Y 559.904,Z 702.53,A -85,B 0,C 180,E1 3036.399,E2 3036.399} C_VEL
LIN {X 0,Y 560.127,Z 702.53,A -85,B 0,C 180,E1 3041.156,E2 3041.156} C_VEL
LIN {X 0,Y 560.295,Z 702.53,A -85,B 0,C 180,E1 3045.988,E2 3045.988} C_VEL
LIN {X 0,Y 560.135,Z 702.53,A -85,B 0,C 180,E1 3052.663,E2 3052.663} C_VEL
LIN {X 0,Y 560.297,Z 702.53,A -85,B 0,C 180,E1 3056.925,E2 3056.925} C_VEL
LIN {X 0,Y 560.458,Z 702.53,A -85,B 0,C 180,E1 3061.555,E2 3061.555} C_VEL
LIN {X 0,Y 560.351,Z 702.53,A -85,B 0,C 180,E1 3066.195,E2 3066.195} C_VEL
LIN {X 0,Y 559.989,Z 702.53,A -85,B 0,C 180,E1 3072.571,E2 3072.571} C_VEL
LIN {X 0,Y 559.987,Z 702.53,A -85,B 0,C 180,E1 3076.047,E2 3076.047} C_VEL
LIN {X 0,Y 555.985,Z 702.53,A -85,B 0,C 180,E1 3077.791,E2 3077.791} C_VEL
LIN {X 0,Y 551.997,Z 702.53,A -85,B 0,C 180,E1 3079.559,E2 3079.559} C_VEL
LIN {X 0,Y 552.031,Z 702.53,A -85,B 0,C 180,E1 3085.566,E2 3085.566} C_VEL
LIN {X 0,Y 551.844,Z 702.53,A -85,B 0,C 180,E1 3091.309,E2 3091.309} C_VEL
LIN {X 0,Y 551.974,Z 702.53,A -85,B 0,C 180,E1 3097.55,E2 3097.55} C_VEL
LIN {X 0,Y 551.957,Z 702.53,A -85,B 0,C 180,E1 3103.121,E2 3103.121} C_VEL
LIN {X 0,Y 551.866,Z 702.53,A -85,B 0,C 180,E1 3108.985,E2 3108.985} C_VEL
LIN {X 0,Y 552,Z 702.53,A -85,B 0,C 180,E1 3115.099,E2 3115.099} C_VEL
LIN {X 0,Y 552.143,Z 702.862,A -85,B 0,C 180,E1 3117.077,E2 3117.077} C_VEL
LIN {X 0,Y 560.667,Z 722.125,A -85,B 0,C 180,E1 3117.925,E2 3117.925} C_VEL
LIN {X 0,Y 560.301,Z 778.21,A -85,B 0,C 180,E1 3118.897,E2 3118.897} C_VEL
LIN {X 0,Y 559.327,Z 817.63,A -85,B 0,C 180,E1 3120.224,E2 3120.224} C_VEL
LIN {X 0,Y 557.929,Z 854.309,A -85,B 0,C 180,E1 3122.089,E2 3122.089} C_VEL
LIN {X 0,Y 556.437,Z 888.988,A -85,B 0,C 180,E1 3124.528,E2 3124.528} C_VEL
LIN {X 0,Y 555.066,Z 920.229,A -85,B 0,C 180,E1 3127.439,E2 3127.439} C_VEL
LIN {X 0,Y 553.915,Z 946.922,A -85,B 0,C 180,E1 3130.667,E2 3130.667} C_VEL
LIN {X 0,Y 553.097,Z 969.169,A -85,B 0,C 180,E1 3134.167,E2 3134.167} C_VEL
LIN {X 0,Y 552.72,Z 986.442,A -85,B 0,C 180,E1 3137.784,E2 3137.784} C_VEL
LIN {X 0,Y 552.595,Z 999.717,A -85,B 0,C 180,E1 3141.757,E2 3141.757} C_VEL
LIN {X 0,Y 552.457,Z 1006.956,A -85,B 0,C 180,E1 3145.299,E2 3145.299} C_VEL
LIN {X 0,Y 552.462,Z 1010.087,A -85,B 0,C 180,E1 3148.435,E2 3148.435} C_VEL
LIN {X 0,Y 552.581,Z 1010.087,A -85,B 0,C 180,E1 3151.565,E2 3151.565} C_VEL
LIN {X 0,Y 552.555,Z 1005.756,A -85,B 0,C 180,E1 3155.485,E2 3155.485} C_VEL
LIN {X 0,Y 552.625,Z 996.303,A -85,B 0,C 180,E1 3159.43,E2 3159.43} C_VEL
LIN {X 0,Y 552.922,Z 981.282,A -85,B 0,C 180,E1 3163.414,E2 3163.414} C_VEL
LIN {X 0,Y 553.487,Z 959.987,A -85,B 0,C 180,E1 3167.402,E2 3167.402} C_VEL
LIN {X 0,Y 554.452,Z 934.613,A -85,B 0,C 180,E1 3170.929,E2 3170.929} C_VEL
LIN {X 0,Y 555.763,Z 903.997,A -85,B 0,C 180,E1 3174.17,E2 3174.17} C_VEL
LIN {X 0,Y 557.19,Z 870.828,A -85,B 0,C 180,E1 3176.839,E2 3176.839} C_VEL
LIN {X 0,Y 558.686,Z 835.801,A -85,B 0,C 180,E1 3178.931,E2 3178.931} C_VEL
LIN {X 0,Y 559.835,Z 799.385,A -85,B 0,C 180,E1 3180.47,E2 3180.47} C_VEL
LIN {X 0,Y 560.735,Z 762.476,A -85,B 0,C 180,E1 3181.442,E2 3181.442} C_VEL
LIN {X 0,Y 560.112,Z 721.015,A -85,B 0,C 180,E1 3182.127,E2 3182.127} C_VEL
LIN {X 0,Y 551.912,Z 702.53,A -85,B 0,C 180,E1 3183.007,E2 3183.007} C_VEL
LIN {X 0,Y 551.947,Z 702.53,A -85,B 0,C 180,E1 3188.963,E2 3188.963} C_VEL
LIN {X 0,Y 551.931,Z 702.53,A -85,B 0,C 180,E1 3194.691,E2 3194.691} C_VEL
LIN {X 0,Y 551.827,Z 702.53,A -85,B 0,C 180,E1 3199.968,E2 3199.968} C_VEL
LIN {X 0,Y 551.968,Z 702.53,A -85,B 0,C 180,E1 3205.101,E2 3205.101} C_VEL
LIN {X 0,Y 552.067,Z 702.53,A -85,B 0,C 180,E1 3211.008,E2 3211.008} C_VEL
LIN {X 0,Y 551.967,Z 702.53,A -85,B 0,C 180,E1 3215.782,E2 3215.782} C_VEL
LIN {X 0,Y 552.117,Z 702.53,A -85,B 0,C 180,E1 3220.845,E2 3220.845} C_VEL
LIN {X 0,Y 552.241,Z 702.53,A -85,B 0,C 180,E1 3225.754,E2 3225.754} C_VEL
LIN {X 0,Y 552.312,Z 702.53,A -85,B 0,C 180,E1 3232.137,E2 3232.137} C_VEL
LIN {X 0,Y 552.423,Z 702.53,A -85,B 0,C 180,E1 3236.856,E2 3236.856} C_VEL
LIN {X 0,Y 552.543,Z 702.53,A -85,B 0,C 180,E1 3241.552,E2 3241.552} C_VEL
LIN {X 0,Y 552.451,Z 702.53,A -85,B 0,C 180,E1 3246.259,E2 3246.259} C_VEL
LIN {X 0,Y 552.123,Z 702.53,A -85,B 0,C 180,E1 3252.614,E2 3252.614} C_VEL
LIN {X 0,Y 552.101,Z 702.53,A -85,B 0,C 180,E1 3257.48,E2 3257.48} C_VEL
LIN {X 0,Y 551.984,Z 702.53,A -85,B 0,C 180,E1 3262.484,E2 3262.484} C_VEL
LIN {X 0,Y 551.875,Z 702.53,A -85,B 0,C 180,E1 3267.679,E2 3267.679} C_VEL
LIN {X 0,Y 551.893,Z 702.53,A -85,B 0,C 180,E1 3273.128,E2 3273.128} C_VEL
LIN {X 0,Y 551.96,Z 702.53,A -85,B 0,C 180,E1 3278.935,E2 3278.935} C_VEL
LIN {X 0,Y 551.93,Z 702.53,A -85,B 0,C 180,E1 3284.695,E2 3284.695} C_VEL
LIN {X 0,Y 551.848,Z 702.53,A -85,B 0,C 180,E1 3289.93,E2 3289.93} C_VEL
LIN {X 0,Y 551.945,Z 702.53,A -85,B 0,C 180,E1 3295.064,E2 3295.064} C_VEL
LIN {X 0,Y 552.072,Z 702.53,A -85,B 0,C 180,E1 3300.957,E2 3300.957} C_VEL
LIN {X 0,Y 552.016,Z 702.53,A -85,B 0,C 180,E1 3305.792,E2 3305.792} C_VEL
LIN {X 0,Y 552.109,Z 702.53,A -85,B 0,C 180,E1 3310.854,E2 3310.854} C_VEL
LIN {X 0,Y 552.245,Z 702.53,A -85,B 0,C 180,E1 3315.764,E2 3315.764} C_VEL
LIN {X 0,Y 552.296,Z 702.53,A -85,B 0,C 180,E1 3322.148,E2 3322.148} C_VEL
LIN {X 0,Y 552.393,Z 702.53,A -85,B 0,C 180,E1 3326.868,E2 3326.868} C_VEL
LIN {X 0,Y 552.027,Z 702.654,A -85,B 0,C 180,E1 3329.247,E2 3329.247} C_VEL
LIN {X 0,Y 558.361,Z 722.038,A -85,B 0,C 180,E1 3329.948,E2 3329.948} C_VEL
LIN {X 0,Y 557.698,Z 759.919,A -85,B 0,C 180,E1 3331.114,E2 3331.114} C_VEL
LIN {X 0,Y 556.529,Z 796.079,A -85,B 0,C 180,E1 3332.914,E2 3332.914} C_VEL
LIN {X 0,Y 555.321,Z 829.065,A -85,B 0,C 180,E1 3335.262,E2 3335.262} C_VEL
LIN {X 0,Y 554.221,Z 859.375,A -85,B 0,C 180,E1 3338.219,E2 3338.219} C_VEL
LIN {X 0,Y 553.473,Z 883.677,A -85,B 0,C 180,E1 3341.415,E2 3341.415} C_VEL
LIN {X 0,Y 552.898,Z 903.649,A -85,B 0,C 180,E1 3344.985,E2 3344.985} C_VEL
LIN {X 0,Y 552.66,Z 918.039,A -85,B 0,C 180,E1 3348.713,E2 3348.713} C_VEL
LIN {X 0,Y 552.479,Z 926.84,A -85,B 0,C 180,E1 3352.482,E2 3352.482} C_VEL
LIN {X 0,Y 552.356,Z 930.284,A -85,B 0,C 180,E1 3355.92,E2 3355.92} C_VEL
LIN {X 0,Y 552.387,Z 929.362,A -85,B 0,C 180,E1 3359.455,E2 3359.455} C_VEL
LIN {X 0,Y 552.526,Z 923.602,A -85,B 0,C 180,E1 3363.109,E2 3363.109} C_VEL
LIN {X 0,Y 552.726,Z 912.114,A -85,B 0,C 180,E1 3366.916,E2 3366.916} C_VEL
LIN {X 0,Y 553.059,Z 895.531,A -85,B 0,C 180,E1 3370.52,E2 3370.52} C_VEL
LIN {X 0,Y 553.811,Z 873.01,A -85,B 0,C 180,E1 3374.021,E2 3374.021} C_VEL
LIN {X 0,Y 554.752,Z 845.222,A -85,B 0,C 180,E1 3377.183,E2 3377.183} C_VEL
LIN {X 0,Y 555.891,Z 813.658,A -85,B 0,C 180,E1 3379.845,E2 3379.845} C_VEL
LIN {X 0,Y 557.087,Z 779.158,A -85,B 0,C 180,E1 3381.928,E2 3381.928} C_VEL
LIN {X 0,Y 558.107,Z 743.084,A -85,B 0,C 180,E1 3383.392,E2 3383.392} C_VEL
LIN {X 0,Y 558.113,Z 718.556,A -85,B 0,C 180,E1 3384.053,E2 3384.053} C_VEL
LIN {X 0,Y 552.086,Z 702.53,A -85,B 0,C 180,E1 3384.738,E2 3384.738} C_VEL
LIN {X 0,Y 552,Z 702.53,A -85,B 0,C 180,E1 3391.022,E2 3391.022} C_VEL
LIN {X 0,Y 551.985,Z 702.53,A -85,B 0,C 180,E1 3395.811,E2 3395.811} C_VEL
LIN {X 0,Y 552.212,Z 702.53,A -85,B 0,C 180,E1 3400.875,E2 3400.875} C_VEL
LIN {X 0,Y 552.376,Z 702.53,A -85,B 0,C 180,E1 3405.783,E2 3405.783} C_VEL
LIN {X 0,Y 552.286,Z 702.53,A -85,B 0,C 180,E1 3412.162,E2 3412.162} C_VEL
LIN {X 0,Y 552.399,Z 702.53,A -85,B 0,C 180,E1 3416.881,E2 3416.881} C_VEL
LIN {X 0,Y 552.549,Z 702.53,A -85,B 0,C 180,E1 3421.577,E2 3421.577} C_VEL
LIN {X 0,Y 552.145,Z 702.53,A -85,B 0,C 180,E1 3427.865,E2 3427.865} C_VEL
LIN {X 0,Y 552.093,Z 702.53,A -85,B 0,C 180,E1 3432.64,E2 3432.64} C_VEL
LIN {X 0,Y 552.047,Z 702.53,A -85,B 0,C 180,E1 3437.508,E2 3437.508} C_VEL
LIN {X 0,Y 551.997,Z 702.53,A -85,B 0,C 180,E1 3439.559,E2 3439.559} C_VEL
LIN {X 0,Y 548.009,Z 702.53,A -85,B 0,C 180,E1 3441.33,E2 3441.33} C_VEL
LIN {X 0,Y 544.03,Z 702.53,A -85,B 0,C 180,E1 3443.126,E2 3443.126} C_VEL
LIN {X 0,Y 543.976,Z 702.53,A -85,B 0,C 180,E1 3448.145,E2 3448.145} C_VEL
LIN {X 0,Y 543.906,Z 702.53,A -85,B 0,C 180,E1 3453.709,E2 3453.709} C_VEL
LIN {X 0,Y 544.014,Z 702.53,A -85,B 0,C 180,E1 3459.647,E2 3459.647} C_VEL
LIN {X 0,Y 543.983,Z 702.53,A -85,B 0,C 180,E1 3463.913,E2 3463.913} C_VEL
LIN {X 0,Y 543.913,Z 702.53,A -85,B 0,C 180,E1 3470.349,E2 3470.349} C_VEL
LIN {X 0,Y 544.172,Z 702.566,A -85,B 0,C 180,E1 3476.528,E2 3476.528} C_VEL
LIN {X 0,Y 554.024,Z 725.212,A -85,B 0,C 180,E1 3477.54,E2 3477.54} C_VEL
LIN {X 0,Y 553.491,Z 779.41,A -85,B 0,C 180,E1 3478.506,E2 3478.506} C_VEL
LIN {X 0,Y 552.392,Z 817.565,A -85,B 0,C 180,E1 3479.809,E2 3479.809} C_VEL
LIN {X 0,Y 550.814,Z 854.385,A -85,B 0,C 180,E1 3481.701,E2 3481.701} C_VEL
LIN {X 0,Y 549.116,Z 889.426,A -85,B 0,C 180,E1 3484.201,E2 3484.201} C_VEL
LIN {X 0,Y 547.577,Z 920.033,A -85,B 0,C 180,E1 3487.091,E2 3487.091} C_VEL
LIN {X 0,Y 546.23,Z 947.339,A -85,B 0,C 180,E1 3490.443,E2 3490.443} C_VEL
LIN {X 0,Y 545.295,Z 970.262,A -85,B 0,C 180,E1 3494.14,E2 3494.14} C_VEL
LIN {X 0,Y 544.83,Z 987.98,A -85,B 0,C 180,E1 3498.011,E2 3498.011} C_VEL
LIN {X 0,Y 544.716,Z 999.717,A -85,B 0,C 180,E1 3501.637,E2 3501.637} C_VEL
LIN {X 0,Y 544.557,Z 1006.956,A -85,B 0,C 180,E1 3505.231,E2 3505.231} C_VEL
LIN {X 0,Y 544.562,Z 1010.087,A -85,B 0,C 180,E1 3508.412,E2 3508.412} C_VEL
LIN {X 0,Y 544.675,Z 1010.088,A -85,B 0,C 180,E1 3511.587,E2 3511.587} C_VEL
LIN {X 0,Y 544.659,Z 1005.756,A -85,B 0,C 180,E1 3515.565,E2 3515.565} C_VEL
LIN {X 0,Y 544.727,Z 996.303,A -85,B 0,C 180,E1 3519.568,E2 3519.568} C_VEL
LIN {X 0,Y 545.069,Z 981.472,A -85,B 0,C 180,E1 3523.566,E2 3523.566} C_VEL
LIN {X 0,Y 545.722,Z 960.81,A -85,B 0,C 180,E1 3527.52,E2 3527.52} C_VEL
LIN {X 0,Y 546.849,Z 934.744,A -85,B 0,C 180,E1 3531.218,E2 3531.218} C_VEL
LIN {X 0,Y 548.361,Z 904.271,A -85,B 0,C 180,E1 3534.492,E2 3534.492} C_VEL
LIN {X 0,Y 549.967,Z 871.092,A -85,B 0,C 180,E1 3537.201,E2 3537.201} C_VEL
LIN {X 0,Y 551.702,Z 835.174,A -85,B 0,C 180,E1 3539.366,E2 3539.366} C_VEL
LIN {X 0,Y 553.009,Z 798.838,A -85,B 0,C 180,E1 3540.906,E2 3540.906} C_VEL
LIN {X 0,Y 553.997,Z 762.431,A -85,B 0,C 180,E1 3541.87,E2 3541.87} C_VEL
LIN {X 0,Y 553.489,Z 723.873,A -85,B 0,C 180,E1 3542.515,E2 3542.515} C_VEL
LIN {X 0,Y 543.955,Z 702.53,A -85,B 0,C 180,E1 3543.543,E2 3543.543} C_VEL
LIN {X 0,Y 544.011,Z 702.53,A -85,B 0,C 180,E1 3549.642,E2 3549.642} C_VEL
LIN {X 0,Y 544.031,Z 702.53,A -85,B 0,C 180,E1 3553.903,E2 3553.903} C_VEL
LIN {X 0,Y 543.905,Z 702.53,A -85,B 0,C 180,E1 3560.343,E2 3560.343} C_VEL
LIN {X 0,Y 544.113,Z 702.53,A -85,B 0,C 180,E1 3566.306,E2 3566.306} C_VEL
LIN {X 0,Y 544.06,Z 702.53,A -85,B 0,C 180,E1 3571.86,E2 3571.86} C_VEL
LIN {X 0,Y 544.043,Z 702.53,A -85,B 0,C 180,E1 3577.142,E2 3577.142} C_VEL
LIN {X 0,Y 544.237,Z 702.53,A -85,B 0,C 180,E1 3582.233,E2 3582.233} C_VEL
LIN {X 0,Y 544.317,Z 702.53,A -85,B 0,C 180,E1 3587.176,E2 3587.176} C_VEL
LIN {X 0,Y 544.394,Z 702.53,A -85,B 0,C 180,E1 3592.022,E2 3592.022} C_VEL
LIN {X 0,Y 544.514,Z 702.53,A -85,B 0,C 180,E1 3596.811,E2 3596.811} C_VEL
LIN {X 0,Y 544.633,Z 702.53,A -85,B 0,C 180,E1 3601.575,E2 3601.575} C_VEL
LIN {X 0,Y 544.52,Z 702.53,A -85,B 0,C 180,E1 3606.35,E2 3606.35} C_VEL
LIN {X 0,Y 544.321,Z 702.53,A -85,B 0,C 180,E1 3611.174,E2 3611.174} C_VEL
LIN {X 0,Y 544.23,Z 702.53,A -85,B 0,C 180,E1 3616.081,E2 3616.081} C_VEL
LIN {X 0,Y 544.154,Z 702.53,A -85,B 0,C 180,E1 3621.113,E2 3621.113} C_VEL
LIN {X 0,Y 544.02,Z 702.53,A -85,B 0,C 180,E1 3626.327,E2 3626.327} C_VEL
LIN {X 0,Y 543.997,Z 702.53,A -85,B 0,C 180,E1 3631.783,E2 3631.783} C_VEL
LIN {X 0,Y 544.07,Z 702.53,A -85,B 0,C 180,E1 3637.577,E2 3637.577} C_VEL
LIN {X 0,Y 544.042,Z 702.53,A -85,B 0,C 180,E1 3643.872,E2 3643.872} C_VEL
LIN {X 0,Y 543.943,Z 702.53,A -85,B 0,C 180,E1 3650.352,E2 3650.352} C_VEL
LIN {X 0,Y 544.072,Z 702.53,A -85,B 0,C 180,E1 3656.309,E2 3656.309} C_VEL
LIN {X 0,Y 544.081,Z 702.53,A -85,B 0,C 180,E1 3661.869,E2 3661.869} C_VEL
LIN {X 0,Y 544.1,Z 702.53,A -85,B 0,C 180,E1 3667.153,E2 3667.153} C_VEL
LIN {X 0,Y 544.239,Z 702.53,A -85,B 0,C 180,E1 3672.242,E2 3672.242} C_VEL
LIN {X 0,Y 544.299,Z 702.53,A -85,B 0,C 180,E1 3677.186,E2 3677.186} C_VEL
LIN {X 0,Y 544.379,Z 702.53,A -85,B 0,C 180,E1 3682.033,E2 3682.033} C_VEL
LIN {X 0,Y 544.486,Z 702.53,A -85,B 0,C 180,E1 3686.823,E2 3686.823} C_VEL
LIN {X 0,Y 544.139,Z 702.582,A -85,B 0,C 180,E1 3688.808,E2 3688.808} C_VEL
LIN {X 0,Y 551.317,Z 723.563,A -85,B 0,C 180,E1 3689.608,E2 3689.608} C_VEL
LIN {X 0,Y 550.492,Z 762.107,A -85,B 0,C 180,E1 3690.846,E2 3690.846} C_VEL
LIN {X 0,Y 549.173,Z 797.438,A -85,B 0,C 180,E1 3692.658,E2 3692.658} C_VEL
LIN {X 0,Y 547.787,Z 830.114,A -85,B 0,C 180,E1 3695.038,E2 3695.038} C_VEL
LIN {X 0,Y 546.613,Z 859.262,A -85,B 0,C 180,E1 3697.934,E2 3697.934} C_VEL
LIN {X 0,Y 545.72,Z 883.502,A -85,B 0,C 180,E1 3701.161,E2 3701.161} C_VEL
LIN {X 0,Y 545.062,Z 903.782,A -85,B 0,C 180,E1 3704.838,E2 3704.838} C_VEL
LIN {X 0,Y 544.799,Z 917.984,A -85,B 0,C 180,E1 3708.575,E2 3708.575} C_VEL
LIN {X 0,Y 544.592,Z 926.489,A -85,B 0,C 180,E1 3712.185,E2 3712.185} C_VEL
LIN {X 0,Y 544.428,Z 929.5,A -85,B 0,C 180,E1 3714.568,E2 3714.568} C_VEL
LIN {X 0,Y 544.418,Z 930.259,A -85,B 0,C 180,E1 3718.113,E2 3718.113} C_VEL
LIN {X 0,Y 544.588,Z 926.422,A -85,B 0,C 180,E1 3721.768,E2 3721.768} C_VEL
LIN {X 0,Y 544.787,Z 917.266,A -85,B 0,C 180,E1 3725.57,E2 3725.57} C_VEL
LIN {X 0,Y 545.005,Z 903.14,A -85,B 0,C 180,E1 3729.207,E2 3729.207} C_VEL
LIN {X 0,Y 545.636,Z 883.725,A -85,B 0,C 180,E1 3732.717,E2 3732.717} C_VEL
LIN {X 0,Y 546.573,Z 858.982,A -85,B 0,C 180,E1 3736.011,E2 3736.011} C_VEL
LIN {X 0,Y 547.892,Z 829.064,A -85,B 0,C 180,E1 3738.957,E2 3738.957} C_VEL
LIN {X 0,Y 549.197,Z 796.971,A -85,B 0,C 180,E1 3741.28,E2 3741.28} C_VEL
LIN {X 0,Y 550.503,Z 763.549,A -85,B 0,C 180,E1 3742.998,E2 3742.998} C_VEL
LIN {X 0,Y 551.564,Z 727.087,A -85,B 0,C 180,E1 3744.206,E2 3744.206} C_VEL
LIN {X 0,Y 550.411,Z 719.056,A -85,B 0,C 180,E1 3744.452,E2 3744.452} C_VEL
LIN {X 0,Y 544.12,Z 702.53,A -85,B 0,C 180,E1 3745.174,E2 3745.174} C_VEL
LIN {X 0,Y 544.018,Z 702.53,A -85,B 0,C 180,E1 3750.069,E2 3750.069} C_VEL
LIN {X 0,Y 544.081,Z 702.53,A -85,B 0,C 180,E1 3755.436,E2 3755.436} C_VEL
LIN {X 0,Y 544.287,Z 702.53,A -85,B 0,C 180,E1 3760.586,E2 3760.586} C_VEL
LIN {X 0,Y 544.454,Z 702.53,A -85,B 0,C 180,E1 3765.948,E2 3765.948} C_VEL
LIN {X 0,Y 544.369,Z 702.53,A -85,B 0,C 180,E1 3772.048,E2 3772.048} C_VEL
LIN {X 0,Y 544.49,Z 702.53,A -85,B 0,C 180,E1 3776.836,E2 3776.836} C_VEL
LIN {X 0,Y 544.638,Z 702.53,A -85,B 0,C 180,E1 3781.6,E2 3781.6} C_VEL
LIN {X 0,Y 544.232,Z 702.53,A -85,B 0,C 180,E1 3787.98,E2 3787.98} C_VEL
LIN {X 0,Y 544.169,Z 702.53,A -85,B 0,C 180,E1 3792.827,E2 3792.827} C_VEL
LIN {X 0,Y 544.116,Z 702.53,A -85,B 0,C 180,E1 3797.771,E2 3797.771} C_VEL
LIN {X 0,Y 544.03,Z 702.53,A -85,B 0,C 180,E1 3803.126,E2 3803.126} C_VEL
LIN {X 0,Y 542.734,Z 702.53,A -85,B 0,C 180,E1 3804.039,E2 3804.039} C_VEL
LIN {X 0,Y 536.154,Z 702.53,A -85,B 0,C 180,E1 3806.524,E2 3806.524} C_VEL
LIN {X 0,Y 536.081,Z 702.53,A -85,B 0,C 180,E1 3806.759,E2 3806.759} C_VEL
LIN {X 0,Y 535.993,Z 702.53,A -85,B 0,C 180,E1 3812.369,E2 3812.369} C_VEL
LIN {X 0,Y 536.146,Z 702.53,A -85,B 0,C 180,E1 3818.264,E2 3818.264} C_VEL
LIN {X 0,Y 535.96,Z 702.53,A -85,B 0,C 180,E1 3824.745,E2 3824.745} C_VEL
LIN {X 0,Y 535.958,Z 702.53,A -85,B 0,C 180,E1 3829.64,E2 3829.64} C_VEL
LIN {X 0,Y 536.191,Z 702.881,A -85,B 0,C 180,E1 3835.967,E2 3835.967} C_VEL
LIN {X 0,Y 547.356,Z 727.234,A -85,B 0,C 180,E1 3837.126,E2 3837.126} C_VEL
LIN {X 0,Y 546.733,Z 779.847,A -85,B 0,C 180,E1 3838.084,E2 3838.084} C_VEL
LIN {X 0,Y 545.489,Z 817.706,A -85,B 0,C 180,E1 3839.393,E2 3839.393} C_VEL
LIN {X 0,Y 543.721,Z 854.609,A -85,B 0,C 180,E1 3841.313,E2 3841.313} C_VEL
LIN {X 0,Y 541.761,Z 889.909,A -85,B 0,C 180,E1 3843.868,E2 3843.868} C_VEL
LIN {X 0,Y 540.071,Z 920.033,A -85,B 0,C 180,E1 3846.754,E2 3846.754} C_VEL
LIN {X 0,Y 538.593,Z 947.34,A -85,B 0,C 180,E1 3850.154,E2 3850.154} C_VEL
LIN {X 0,Y 537.481,Z 970.263,A -85,B 0,C 180,E1 3853.904,E2 3853.904} C_VEL
LIN {X 0,Y 537.034,Z 986.443,A -85,B 0,C 180,E1 3857.422,E2 3857.422} C_VEL
LIN {X 0,Y 536.816,Z 999.717,A -85,B 0,C 180,E1 3861.513,E2 3861.513} C_VEL
LIN {X 0,Y 536.659,Z 1006.956,A -85,B 0,C 180,E1 3865.161,E2 3865.161} C_VEL
LIN {X 0,Y 536.672,Z 1010.087,A -85,B 0,C 180,E1 3868.389,E2 3868.389} C_VEL
LIN {X 0,Y 536.799,Z 1010.088,A -85,B 0,C 180,E1 3871.611,E2 3871.611} C_VEL
LIN {X 0,Y 536.762,Z 1005.756,A -85,B 0,C 180,E1 3875.647,E2 3875.647} C_VEL
LIN {X 0,Y 536.837,Z 996.304,A -85,B 0,C 180,E1 3879.71,E2 3879.71} C_VEL
LIN {X 0,Y 537.256,Z 980.778,A -85,B 0,C 180,E1 3883.932,E2 3883.932} C_VEL
LIN {X 0,Y 538.058,Z 959.665,A -85,B 0,C 180,E1 3887.969,E2 3887.969} C_VEL
LIN {X 0,Y 539.337,Z 933.554,A -85,B 0,C 180,E1 3891.675,E2 3891.675} C_VEL
LIN {X 0,Y 540.999,Z 903.325,A -85,B 0,C 180,E1 3894.939,E2 3894.939} C_VEL
LIN {X 0,Y 542.859,Z 869.608,A -85,B 0,C 180,E1 3897.696,E2 3897.696} C_VEL
LIN {X 0,Y 544.719,Z 834.365,A -85,B 0,C 180,E1 3899.823,E2 3899.823} C_VEL
LIN {X 0,Y 546.251,Z 796.842,A -85,B 0,C 180,E1 3901.402,E2 3901.402} C_VEL
LIN {X 0,Y 547.339,Z 760.646,A -85,B 0,C 180,E1 3902.336,E2 3902.336} C_VEL
LIN {X 0,Y 546.787,Z 726.446,A -85,B 0,C 180,E1 3902.925,E2 3902.925} C_VEL
LIN {X 0,Y 536.004,Z 702.53,A -85,B 0,C 180,E1 3904.094,E2 3904.094} C_VEL
LIN {X 0,Y 536.138,Z 702.53,A -85,B 0,C 180,E1 3908.259,E2 3908.259} C_VEL
LIN {X 0,Y 536.005,Z 702.53,A -85,B 0,C 180,E1 3914.735,E2 3914.735} C_VEL
LIN {X 0,Y 535.957,Z 702.53,A -85,B 0,C 180,E1 3919.635,E2 3919.635} C_VEL
LIN {X 0,Y 536.096,Z 702.53,A -85,B 0,C 180,E1 3925.732,E2 3925.732} C_VEL
LIN {X 0,Y 536.114,Z 702.53,A -85,B 0,C 180,E1 3931.405,E2 3931.405} C_VEL
LIN {X 0,Y 536.126,Z 702.53,A -85,B 0,C 180,E1 3936.785,E2 3936.785} C_VEL
LIN {X 0,Y 536.303,Z 702.53,A -85,B 0,C 180,E1 3941.961,E2 3941.961} C_VEL
LIN {X 0,Y 536.435,Z 702.53,A -85,B 0,C 180,E1 3946.984,E2 3946.984} C_VEL
LIN {X 0,Y 536.476,Z 702.53,A -85,B 0,C 180,E1 3951.904,E2 3951.904} C_VEL
LIN {X 0,Y 536.622,Z 702.53,A -85,B 0,C 180,E1 3956.764,E2 3956.764} C_VEL
LIN {X 0,Y 536.731,Z 702.53,A -85,B 0,C 180,E1 3961.598,E2 3961.598} C_VEL
LIN {X 0,Y 536.591,Z 702.53,A -85,B 0,C 180,E1 3966.444,E2 3966.444} C_VEL
LIN {X 0,Y 536.404,Z 702.53,A -85,B 0,C 180,E1 3971.341,E2 3971.341} C_VEL
LIN {X 0,Y 536.257,Z 702.53,A -85,B 0,C 180,E1 3976.911,E2 3976.911} C_VEL
LIN {X 0,Y 536.182,Z 702.53,A -85,B 0,C 180,E1 3981.76,E2 3981.76} C_VEL
LIN {X 0,Y 536.077,Z 702.53,A -85,B 0,C 180,E1 3986.747,E2 3986.747} C_VEL
LIN {X 0,Y 536.028,Z 702.53,A -85,B 0,C 180,E1 3992.376,E2 3992.376} C_VEL
LIN {X 0,Y 536.13,Z 702.53,A -85,B 0,C 180,E1 3998.232,E2 3998.232} C_VEL
LIN {X 0,Y 536.065,Z 702.53,A -85,B 0,C 180,E1 4002.954,E2 4002.954} C_VEL
LIN {X 0,Y 535.964,Z 702.53,A -85,B 0,C 180,E1 4009.445,E2 4009.445} C_VEL
LIN {X 0,Y 536.02,Z 702.53,A -85,B 0,C 180,E1 4014.686,E2 4014.686} C_VEL
LIN {X 0,Y 536.182,Z 702.53,A -85,B 0,C 180,E1 4019.563,E2 4019.563} C_VEL
LIN {X 0,Y 536.133,Z 702.53,A -85,B 0,C 180,E1 4025.027,E2 4025.027} C_VEL
LIN {X 0,Y 536.248,Z 702.53,A -85,B 0,C 180,E1 4030.264,E2 4030.264} C_VEL
LIN {X 0,Y 536.365,Z 702.53,A -85,B 0,C 180,E1 4035.333,E2 4035.333} C_VEL
LIN {X 0,Y 536.462,Z 702.53,A -85,B 0,C 180,E1 4041.915,E2 4041.915} C_VEL
LIN {X 0,Y 536.371,Z 702.53,A -85,B 0,C 180,E1 4047.582,E2 4047.582} C_VEL
LIN {X 0,Y 536.274,Z 702.53,A -85,B 0,C 180,E1 4048.337,E2 4048.337} C_VEL
LIN {X 0,Y 544.285,Z 726.452,A -85,B 0,C 180,E1 4049.291,E2 4049.291} C_VEL
LIN {X 0,Y 543.282,Z 763.712,A -85,B 0,C 180,E1 4050.547,E2 4050.547} C_VEL
LIN {X 0,Y 541.822,Z 798.801,A -85,B 0,C 180,E1 4052.395,E2 4052.395} C_VEL
LIN {X 0,Y 540.222,Z 832.296,A -85,B 0,C 180,E1 4054.908,E2 4054.908} C_VEL
LIN {X 0,Y 538.847,Z 861.5,A -85,B 0,C 180,E1 4057.921,E2 4057.921} C_VEL
LIN {X 0,Y 537.865,Z 886.048,A -85,B 0,C 180,E1 4061.326,E2 4061.326} C_VEL
LIN {X 0,Y 537.157,Z 905.55,A -85,B 0,C 180,E1 4065.062,E2 4065.062} C_VEL
LIN {X 0,Y 536.865,Z 919.136,A -85,B 0,C 180,E1 4068.859,E2 4068.859} C_VEL
LIN {X 0,Y 536.709,Z 926.253,A -85,B 0,C 180,E1 4071.968,E2 4071.968} C_VEL
LIN {X 0,Y 536.485,Z 930.283,A -85,B 0,C 180,E1 4075.887,E2 4075.887} C_VEL
LIN {X 0,Y 536.538,Z 929.502,A -85,B 0,C 180,E1 4079.373,E2 4079.373} C_VEL
LIN {X 0,Y 536.784,Z 923.501,A -85,B 0,C 180,E1 4083.333,E2 4083.333} C_VEL
LIN {X 0,Y 537.003,Z 912.081,A -85,B 0,C 180,E1 4087.219,E2 4087.219} C_VEL
LIN {X 0,Y 537.537,Z 894.699,A -85,B 0,C 180,E1 4091.079,E2 4091.079} C_VEL
LIN {X 0,Y 538.429,Z 871.809,A -85,B 0,C 180,E1 4094.685,E2 4094.685} C_VEL
LIN {X 0,Y 539.648,Z 845.106,A -85,B 0,C 180,E1 4097.786,E2 4097.786} C_VEL
LIN {X 0,Y 541.142,Z 813.512,A -85,B 0,C 180,E1 4100.516,E2 4100.516} C_VEL
LIN {X 0,Y 542.694,Z 778.62,A -85,B 0,C 180,E1 4102.666,E2 4102.666} C_VEL
LIN {X 0,Y 544.005,Z 742.536,A -85,B 0,C 180,E1 4104.151,E2 4104.151} C_VEL
LIN {X 0,Y 544.077,Z 723.097,A -85,B 0,C 180,E1 4104.707,E2 4104.707} C_VEL
LIN {X 0,Y 536.158,Z 702.53,A -85,B 0,C 180,E1 4105.646,E2 4105.646} C_VEL
LIN {X 0,Y 536.113,Z 702.53,A -85,B 0,C 180,E1 4111.434,E2 4111.434} C_VEL
LIN {X 0,Y 536.169,Z 702.53,A -85,B 0,C 180,E1 4116.815,E2 4116.815} C_VEL
LIN {X 0,Y 536.367,Z 702.53,A -85,B 0,C 180,E1 4121.99,E2 4121.99} C_VEL
LIN {X 0,Y 536.495,Z 702.53,A -85,B 0,C 180,E1 4127.012,E2 4127.012} C_VEL
LIN {X 0,Y 536.377,Z 702.53,A -85,B 0,C 180,E1 4132.644,E2 4132.644} C_VEL
LIN {X 0,Y 536.393,Z 702.53,A -85,B 0,C 180,E1 4138.401,E2 4138.401} C_VEL
LIN {X 0,Y 536.462,Z 702.53,A -85,B 0,C 180,E1 4143.237,E2 4143.237} C_VEL
LIN {X 0,Y 536.32,Z 702.53,A -85,B 0,C 180,E1 4148.099,E2 4148.099} C_VEL
LIN {X 0,Y 536.255,Z 702.53,A -85,B 0,C 180,E1 4153.02,E2 4153.02} C_VEL
LIN {X 0,Y 536.204,Z 702.53,A -85,B 0,C 180,E1 4158.042,E2 4158.042} C_VEL
LIN {X 0,Y 536.129,Z 702.53,A -85,B 0,C 180,E1 4163.215,E2 4163.215} C_VEL
LIN {X 0,Y 536.081,Z 702.53,A -85,B 0,C 180,E1 4166.759,E2 4166.759} C_VEL
LIN {X 0,Y 533.552,Z 702.53,A -85,B 0,C 180,E1 4168.139,E2 4168.139} C_VEL
LIN {X 0,Y 528.112,Z 702.53,A -85,B 0,C 180,E1 4170.207,E2 4170.207} C_VEL
LIN {X 0,Y 528.028,Z 702.53,A -85,B 0,C 180,E1 4170.446,E2 4170.446} C_VEL
LIN {X 0,Y 528.188,Z 702.53,A -85,B 0,C 180,E1 4176.874,E2 4176.874} C_VEL
LIN {X 0,Y 528.067,Z 702.53,A -85,B 0,C 180,E1 4183.306,E2 4183.306} C_VEL
LIN {X 0,Y 527.989,Z 702.53,A -85,B 0,C 180,E1 4188.901,E2 4188.901} C_VEL
LIN {X 0,Y 528.221,Z 702.53,A -85,B 0,C 180,E1 4195.365,E2 4195.365} C_VEL
LIN {X 0,Y 540.723,Z 731.398,A -85,B 0,C 180,E1 4196.735,E2 4196.735} C_VEL
LIN {X 0,Y 539.993,Z 780.579,A -85,B 0,C 180,E1 4197.659,E2 4197.659} C_VEL
LIN {X 0,Y 538.616,Z 817.885,A -85,B 0,C 180,E1 4198.968,E2 4198.968} C_VEL
LIN {X 0,Y 536.64,Z 854.795,A -85,B 0,C 180,E1 4200.911,E2 4200.911} C_VEL
LIN {X 0,Y 534.484,Z 889.91,A -85,B 0,C 180,E1 4203.485,E2 4203.485} C_VEL
LIN {X 0,Y 532.489,Z 921.944,A -85,B 0,C 180,E1 4206.625,E2 4206.625} C_VEL
LIN {X 0,Y 530.856,Z 948.704,A -85,B 0,C 180,E1 4210.055,E2 4210.055} C_VEL
LIN {X 0,Y 529.677,Z 971.351,A -85,B 0,C 180,E1 4213.872,E2 4213.872} C_VEL
LIN {X 0,Y 529.131,Z 987.981,A -85,B 0,C 180,E1 4217.649,E2 4217.649} C_VEL
LIN {X 0,Y 528.923,Z 999.717,A -85,B 0,C 180,E1 4221.385,E2 4221.385} C_VEL
LIN {X 0,Y 528.772,Z 1006.957,A -85,B 0,C 180,E1 4225.088,E2 4225.088} C_VEL
LIN {X 0,Y 528.77,Z 1010.087,A -85,B 0,C 180,E1 4228.364,E2 4228.364} C_VEL
LIN {X 0,Y 528.756,Z 1009.406,A -85,B 0,C 180,E1 4232.733,E2 4232.733} C_VEL
LIN {X 0,Y 528.86,Z 1004.223,A -85,B 0,C 180,E1 4236.553,E2 4236.553} C_VEL
LIN {X 0,Y 528.965,Z 994.398,A -85,B 0,C 180,E1 4240.48,E2 4240.48} C_VEL
LIN {X 0,Y 529.501,Z 979.174,A -85,B 0,C 180,E1 4244.498,E2 4244.498} C_VEL
LIN {X 0,Y 530.411,Z 958.342,A -85,B 0,C 180,E1 4248.452,E2 4248.452} C_VEL
LIN {X 0,Y 531.814,Z 932.651,A -85,B 0,C 180,E1 4252.111,E2 4252.111} C_VEL
LIN {X 0,Y 533.621,Z 903.609,A -85,B 0,C 180,E1 4255.28,E2 4255.28} C_VEL
LIN {X 0,Y 535.668,Z 870.459,A -85,B 0,C 180,E1 4258.037,E2 4258.037} C_VEL
LIN {X 0,Y 537.714,Z 835.872,A -85,B 0,C 180,E1 4260.17,E2 4260.17} C_VEL
LIN {X 0,Y 539.403,Z 798.912,A -85,B 0,C 180,E1 4261.773,E2 4261.773} C_VEL
LIN {X 0,Y 540.662,Z 761.006,A -85,B 0,C 180,E1 4262.779,E2 4262.779} C_VEL
LIN {X 0,Y 540.123,Z 728.762,A -85,B 0,C 180,E1 4263.347,E2 4263.347} C_VEL
LIN {X 0,Y 528.099,Z 702.53,A -85,B 0,C 180,E1 4264.722,E2 4264.722} C_VEL
LIN {X 0,Y 528.106,Z 702.53,A -85,B 0,C 180,E1 4269.507,E2 4269.507} C_VEL
LIN {X 0,Y 528.071,Z 702.53,A -85,B 0,C 180,E1 4275.594,E2 4275.594} C_VEL
LIN {X 0,Y 527.989,Z 702.53,A -85,B 0,C 180,E1 4281.034,E2 4281.034} C_VEL
LIN {X 0,Y 528.221,Z 702.53,A -85,B 0,C 180,E1 4287.119,E2 4287.119} C_VEL
LIN {X 0,Y 528.145,Z 702.53,A -85,B 0,C 180,E1 4292.789,E2 4292.789} C_VEL
LIN {X 0,Y 528.224,Z 702.53,A -85,B 0,C 180,E1 4298.19,E2 4298.19} C_VEL
LIN {X 0,Y 528.395,Z 702.53,A -85,B 0,C 180,E1 4303.396,E2 4303.396} C_VEL
LIN {X 0,Y 528.435,Z 702.53,A -85,B 0,C 180,E1 4308.459,E2 4308.459} C_VEL
LIN {X 0,Y 528.537,Z 702.53,A -85,B 0,C 180,E1 4313.431,E2 4313.431} C_VEL
LIN {X 0,Y 528.523,Z 702.53,A -85,B 0,C 180,E1 4318.351,E2 4318.351} C_VEL
LIN {X 0,Y 528.575,Z 702.53,A -85,B 0,C 180,E1 4323.259,E2 4323.259} C_VEL
LIN {X 0,Y 528.448,Z 702.53,A -85,B 0,C 180,E1 4328.193,E2 4328.193} C_VEL
LIN {X 0,Y 528.352,Z 702.53,A -85,B 0,C 180,E1 4333.815,E2 4333.815} C_VEL
LIN {X 0,Y 528.351,Z 702.53,A -85,B 0,C 180,E1 4339.522,E2 4339.522} C_VEL
LIN {X 0,Y 528.193,Z 702.53,A -85,B 0,C 180,E1 4345.354,E2 4345.354} C_VEL
LIN {X 0,Y 528.081,Z 702.53,A -85,B 0,C 180,E1 4350.989,E2 4350.989} C_VEL
LIN {X 0,Y 528.147,Z 702.53,A -85,B 0,C 180,E1 4356.868,E2 4356.868} C_VEL
LIN {X 0,Y 528.127,Z 702.53,A -85,B 0,C 180,E1 4362.021,E2 4362.021} C_VEL
LIN {X 0,Y 527.991,Z 702.53,A -85,B 0,C 180,E1 4367.961,E2 4367.961} C_VEL
LIN {X 0,Y 528.081,Z 702.53,A -85,B 0,C 180,E1 4373.124,E2 4373.124} C_VEL
LIN {X 0,Y 528.215,Z 702.53,A -85,B 0,C 180,E1 4379.054,E2 4379.054} C_VEL
LIN {X 0,Y 528.203,Z 702.53,A -85,B 0,C 180,E1 4384.626,E2 4384.626} C_VEL
LIN {X 0,Y 528.336,Z 702.53,A -85,B 0,C 180,E1 4390.405,E2 4390.405} C_VEL
LIN {X 0,Y 528.478,Z 702.53,A -85,B 0,C 180,E1 4396.795,E2 4396.795} C_VEL
LIN {X 0,Y 528.572,Z 702.53,A -85,B 0,C 180,E1 4401.793,E2 4401.793} C_VEL
LIN {X 0,Y 528.591,Z 702.53,A -85,B 0,C 180,E1 4407.096,E2 4407.096} C_VEL
LIN {X 0,Y 528.453,Z 703.151,A -85,B 0,C 180,E1 4407.886,E2 4407.886} C_VEL
LIN {X 0,Y 537.248,Z 727.929,A -85,B 0,C 180,E1 4408.939,E2 4408.939} C_VEL
LIN {X 0,Y 536.109,Z 765.03,A -85,B 0,C 180,E1 4410.227,E2 4410.227} C_VEL
LIN {X 0,Y 534.483,Z 800.164,A -85,B 0,C 180,E1 4412.124,E2 4412.124} C_VEL
LIN {X 0,Y 532.691,Z 833.266,A -85,B 0,C 180,E1 4414.672,E2 4414.672} C_VEL
LIN {X 0,Y 531.184,Z 862.47,A -85,B 0,C 180,E1 4417.755,E2 4417.755} C_VEL
LIN {X 0,Y 530.063,Z 886.962,A -85,B 0,C 180,E1 4421.24,E2 4421.24} C_VEL
LIN {X 0,Y 529.321,Z 905.485,A -85,B 0,C 180,E1 4424.867,E2 4424.867} C_VEL
LIN {X 0,Y 529.02,Z 918.914,A -85,B 0,C 180,E1 4428.659,E2 4428.659} C_VEL
LIN {X 0,Y 528.756,Z 926.891,A -85,B 0,C 180,E1 4432.316,E2 4432.316} C_VEL
LIN {X 0,Y 528.582,Z 930.036,A -85,B 0,C 180,E1 4435.355,E2 4435.355} C_VEL
LIN {X 0,Y 528.636,Z 929.738,A -85,B 0,C 180,E1 4439.031,E2 4439.031} C_VEL
LIN {X 0,Y 528.838,Z 924.716,A -85,B 0,C 180,E1 4442.831,E2 4442.831} C_VEL
LIN {X 0,Y 529.069,Z 914.145,A -85,B 0,C 180,E1 4446.796,E2 4446.796} C_VEL
LIN {X 0,Y 529.545,Z 898.188,A -85,B 0,C 180,E1 4450.619,E2 4450.619} C_VEL
LIN {X 0,Y 530.476,Z 877.347,A -85,B 0,C 180,E1 4454.163,E2 4454.163} C_VEL
LIN {X 0,Y 531.763,Z 851.703,A -85,B 0,C 180,E1 4457.401,E2 4457.401} C_VEL
LIN {X 0,Y 533.421,Z 820.983,A -85,B 0,C 180,E1 4460.282,E2 4460.282} C_VEL
LIN {X 0,Y 535.106,Z 787.034,A -85,B 0,C 180,E1 4462.581,E2 4462.581} C_VEL
LIN {X 0,Y 536.639,Z 751.676,A -85,B 0,C 180,E1 4464.224,E2 4464.224} C_VEL
LIN {X 0,Y 536.817,Z 724.783,A -85,B 0,C 180,E1 4465.077,E2 4465.077} C_VEL
LIN {X 0,Y 528.213,Z 702.53,A -85,B 0,C 180,E1 4466.142,E2 4466.142} C_VEL
LIN {X 0,Y 528.186,Z 702.53,A -85,B 0,C 180,E1 4472.334,E2 4472.334} C_VEL
LIN {X 0,Y 528.325,Z 702.53,A -85,B 0,C 180,E1 4478.223,E2 4478.223} C_VEL
LIN {X 0,Y 528.476,Z 702.53,A -85,B 0,C 180,E1 4483.426,E2 4483.426} C_VEL
LIN {X 0,Y 528.466,Z 702.53,A -85,B 0,C 180,E1 4488.486,E2 4488.486} C_VEL
LIN {X 0,Y 528.513,Z 702.53,A -85,B 0,C 180,E1 4493.457,E2 4493.457} C_VEL
LIN {X 0,Y 528.493,Z 702.53,A -85,B 0,C 180,E1 4498.377,E2 4498.377} C_VEL
LIN {X 0,Y 528.577,Z 702.53,A -85,B 0,C 180,E1 4503.286,E2 4503.286} C_VEL
LIN {X 0,Y 528.424,Z 702.53,A -85,B 0,C 180,E1 4508.22,E2 4508.22} C_VEL
LIN {X 0,Y 528.309,Z 702.53,A -85,B 0,C 180,E1 4513.795,E2 4513.795} C_VEL
LIN {X 0,Y 528.257,Z 702.53,A -85,B 0,C 180,E1 4519.492,E2 4519.492} C_VEL
LIN {X 0,Y 528.2,Z 702.53,A -85,B 0,C 180,E1 4525.383,E2 4525.383} C_VEL
LIN {X 0,Y 528.028,Z 702.53,A -85,B 0,C 180,E1 4530.446,E2 4530.446} C_VEL
LIN {X 0,Y 525.541,Z 702.53,A -85,B 0,C 180,E1 4531.848,E2 4531.848} C_VEL
LIN {X 0,Y 520.165,Z 702.53,A -85,B 0,C 180,E1 4533.95,E2 4533.95} C_VEL
LIN {X 0,Y 520.063,Z 702.53,A -85,B 0,C 180,E1 4534.193,E2 4534.193} C_VEL
LIN {X 0,Y 520.218,Z 702.53,A -85,B 0,C 180,E1 4539.661,E2 4539.661} C_VEL
LIN {X 0,Y 520.094,Z 702.53,A -85,B 0,C 180,E1 4545.865,E2 4545.865} C_VEL
LIN {X 0,Y 520.066,Z 702.53,A -85,B 0,C 180,E1 4551.58,E2 4551.58} C_VEL
LIN {X 0,Y 520.23,Z 702.67,A -85,B 0,C 180,E1 4554.768,E2 4554.768} C_VEL
LIN {X 0,Y 534.099,Z 732.203,A -85,B 0,C 180,E1 4556.281,E2 4556.281} C_VEL
LIN {X 0,Y 533.302,Z 780.638,A -85,B 0,C 180,E1 4557.205,E2 4557.205} C_VEL
LIN {X 0,Y 531.784,Z 817.633,A -85,B 0,C 180,E1 4558.512,E2 4558.512} C_VEL
LIN {X 0,Y 529.618,Z 854.792,A -85,B 0,C 180,E1 4560.488,E2 4560.488} C_VEL
LIN {X 0,Y 527.26,Z 889.903,A -85,B 0,C 180,E1 4563.092,E2 4563.092} C_VEL
LIN {X 0,Y 525.131,Z 920.162,A -85,B 0,C 180,E1 4566.068,E2 4566.068} C_VEL
LIN {X 0,Y 523.32,Z 947.425,A -85,B 0,C 180,E1 4569.562,E2 4569.562} C_VEL
LIN {X 0,Y 521.99,Z 970.266,A -85,B 0,C 180,E1 4573.412,E2 4573.412} C_VEL
LIN {X 0,Y 521.288,Z 987.982,A -85,B 0,C 180,E1 4577.46,E2 4577.46} C_VEL
LIN {X 0,Y 521.053,Z 999.717,A -85,B 0,C 180,E1 4581.254,E2 4581.254} C_VEL
LIN {X 0,Y 520.876,Z 1006.957,A -85,B 0,C 180,E1 4585.014,E2 4585.014} C_VEL
LIN {X 0,Y 520.885,Z 1010.088,A -85,B 0,C 180,E1 4588.34,E2 4588.34} C_VEL
LIN {X 0,Y 520.998,Z 1010.088,A -85,B 0,C 180,E1 4591.66,E2 4591.66} C_VEL
LIN {X 0,Y 521.001,Z 1005.755,A -85,B 0,C 180,E1 4595.818,E2 4595.818} C_VEL
LIN {X 0,Y 521.098,Z 996.125,A -85,B 0,C 180,E1 4600.072,E2 4600.072} C_VEL
LIN {X 0,Y 521.577,Z 981.346,A -85,B 0,C 180,E1 4604.221,E2 4604.221} C_VEL
LIN {X 0,Y 522.557,Z 961.267,A -85,B 0,C 180,E1 4608.241,E2 4608.241} C_VEL
LIN {X 0,Y 524.178,Z 934.311,A -85,B 0,C 180,E1 4612.238,E2 4612.238} C_VEL
LIN {X 0,Y 526.193,Z 904.811,A -85,B 0,C 180,E1 4615.543,E2 4615.543} C_VEL
LIN {X 0,Y 528.503,Z 871.206,A -85,B 0,C 180,E1 4618.395,E2 4618.395} C_VEL
LIN {X 0,Y 530.848,Z 835.022,A -85,B 0,C 180,E1 4620.648,E2 4620.648} C_VEL
LIN {X 0,Y 532.701,Z 797.789,A -85,B 0,C 180,E1 4622.261,E2 4622.261} C_VEL
LIN {X 0,Y 534.057,Z 759.075,A -85,B 0,C 180,E1 4623.272,E2 4623.272} C_VEL
LIN {X 0,Y 533.5,Z 731.391,A -85,B 0,C 180,E1 4623.775,E2 4623.775} C_VEL
LIN {X 0,Y 520.157,Z 702.53,A -85,B 0,C 180,E1 4625.289,E2 4625.289} C_VEL
LIN {X 0,Y 520.19,Z 702.53,A -85,B 0,C 180,E1 4631.037,E2 4631.037} C_VEL
LIN {X 0,Y 520.12,Z 702.53,A -85,B 0,C 180,E1 4636.496,E2 4636.496} C_VEL
LIN {X 0,Y 520.063,Z 702.53,A -85,B 0,C 180,E1 4642.452,E2 4642.452} C_VEL
LIN {X 0,Y 520.298,Z 702.53,A -85,B 0,C 180,E1 4648.522,E2 4648.522} C_VEL
LIN {X 0,Y 520.23,Z 702.53,A -85,B 0,C 180,E1 4654.2,E2 4654.2} C_VEL
LIN {X 0,Y 520.349,Z 702.53,A -85,B 0,C 180,E1 4659.626,E2 4659.626} C_VEL
LIN {X 0,Y 520.517,Z 702.53,A -85,B 0,C 180,E1 4664.865,E2 4664.865} C_VEL
LIN {X 0,Y 520.629,Z 702.53,A -85,B 0,C 180,E1 4670.223,E2 4670.223} C_VEL
LIN {X 0,Y 520.832,Z 702.53,A -85,B 0,C 180,E1 4676.665,E2 4676.665} C_VEL
LIN {X 0,Y 520.926,Z 702.53,A -85,B 0,C 180,E1 4681.646,E2 4681.646} C_VEL
LIN {X 0,Y 520.739,Z 702.53,A -85,B 0,C 180,E1 4686.641,E2 4686.641} C_VEL
LIN {X 0,Y 520.553,Z 702.53,A -85,B 0,C 180,E1 4691.691,E2 4691.691} C_VEL
